Universal Robots URScript: faichun_9jan_1.script

def faichun_9jan_1():
  set_target_payload(1.070000, [0.002000, 0.003000, 0.057000], [0.001723, 0.001723, 0.001723, 0.000000, 0.000000, 0.000000])
  set_tcp(p[0.0,0.0,0.0,0.0,0.0,0.0])
  set_tool_communication(True, 1000000, 2, 1, 1.5, 3.5)
  set_tool_output_mode(0)
  set_tool_digital_output_mode(0, 1)
  set_tool_digital_output_mode(1, 1)
  set_tool_voltage(24)
  step_count_5365f4e1_2aa6_4e7d_952d_8f9d08daece7 = 0.0
  thread Step_Counter_Thread_19057cb8_9120_4cdd_987b_3fe53dc553a4():
    while (True):
      step_count_5365f4e1_2aa6_4e7d_952d_8f9d08daece7 = step_count_5365f4e1_2aa6_4e7d_952d_8f9d08daece7 + 1.0
      sync()
    end
  end
  run Step_Counter_Thread_19057cb8_9120_4cdd_987b_3fe53dc553a4()
  set_safety_mode_transition_hardness(1)
  set_standard_analog_input_domain(0, 1)
  set_standard_analog_input_domain(1, 1)
  set_tool_analog_input_domain(0, 1)
  set_tool_analog_input_domain(1, 1)
  set_analog_outputdomain(0, 0)
  set_analog_outputdomain(1, 0)
  set_input_actions_to_default()
  set_gravity([0.0, 0.0, 9.82])
  global B1empty=False
  global A2Empty=0
  global A1Empty=0
  global B2Empty=False
  global pallet_step=0
  global bright_box=0
  global Pallet_1_cnt=2
  global dark_boxes=0
  global Point_1=p[0.6913645118948067,-0.12399382748223003,0.49223711947071,-1.2983729986843258,1.1259514972191385,-1.2203503861141718]
  # begin: URCap Installation Node
  #   Source: External Control, 1.0.5, FZI Research Center for Information Technology
  #   Type: External Control
  # end: URCap Installation Node
  # begin: URCap Installation Node
  #   Source: OnRobot, 6.2.0, OnRobot A/S
  #   Type: OnRobot Setup
  sleep(1)
  if (False):
  end
  ON_CONN_SHIFT_BOOL = 64
  ON_CONN_SHIFT_INT = 24
  ON_CONN_SHIFT_FLOAT = 24
  ON_CONN_REG_SUM_BOOL = 0
  ON_CONN_REG_SUM_INT = 1
  ON_CONN_REG_SUM_FLOAT = 0
  ON_TOOL_SHIFT_BOOL = 64
  ON_TOOL_SHIFT_INT = 25
  ON_TOOL_SHIFT_FLOAT = 24
  ON_TOOL_SHIFT_BOOL_ARR = [64, 64, 64]
  ON_TOOL_SHIFT_INT_ARR = [25, 25, 25]
  ON_TOOL_SHIFT_FLOAT_ARR = [24, 24, 24]
  ON_TOOL_REG_SUM_BOOL = 0
  ON_TOOL_REG_SUM_INT = 0
  ON_TOOL_REG_SUM_FLOAT = 0
  ON_REGISTERS_SPEEDL_FLOAT = 0
  ON_REG_USE_TOOL = False
  ON_DI_SINGLE = 0
  ON_DI_PRIMARY = 1
  ON_DI_SECONDARY = 2
  ON_DI_DUAL = 3
  on_robot_type = 10
  on_robot_cycle = 2.0
  on_conn_ip = "localhost"
  on_tool_ip = "localhost"
  on_device_socket_port = 51234
  on_conn_xmlrpc = rpc_factory("xmlrpc", "http://localhost:41414")
  on_tool_xmlrpc = rpc_factory("xmlrpc", "http://localhost:41414")
  on_RPC = rpc_factory("xmlrpc", "http://127.0.0.1:31416")
  ON_DEBUG_LOG = False
  on_isMetric = True
  on_toolConnector = True
  on_ioqc = False
  on_dual = False
  on_computebox = False
  on_devices = 0
  on_gripper = [False, False, False]
  on_custom_tcp_id = "none"
  on_custom_tcp_enabled = False
  speedlTime = 0.001
  on_ft = False
  #======    OnRobot Globals    ======#

  ON_MATH_PI=3.141593
  ON_ZEROPOSE=p[0.0,0.0,0.0,0.0,0.0,0.0]
  ON_ZEROFRAME=p[0.0,0.0,0.0,0.0,0.0,0.0]
  ON_ZERO3D=[0.0,0.0,0.0]
  ON_ZERO6D=[0.0,0.0,0.0,0.0,0.0,0.0]
  ON_ZERO8D=[0.0,0.0,0.0,0.0,0.0,0.0,0.0,0.0]
  ON_FALSE3D=[False,False,False]
  ON_FALSE6D=[False,False,False,False,False,False]
  ON_FALSE8D=[False,False,False,False,False,False,False,False]
  global on_return=0
  on_speedL=ON_ZERO6D
  on_speedBase=ON_ZERO6D
  on_speedVect=ON_ZERO6D
  on_speedExtra=ON_ZERO6D
  on_speedCB=ON_ZERO6D
  on_speedGecko=ON_ZERO6D
  on_RTDE_error=0
  on_RTDE_tool_error=0
  on_dataProcess_thrd=0
  ON_DEVICE_ID_MISSING=0
  ON_INIT_WATCHDOG_HZ=5
  ON_INIT_TIMEOUT=2000
  on_robot_TCP_offset=ON_ZEROFRAME
  on_tcp_offset_actual=ON_ZEROFRAME
  on_cog_actual=ON_ZEROFRAME
  on_mass_actual=0.0
  on_robot_mount=[0.0,0.0]

  #======    End of OnRobot Globals    ======#
  #======    OnRobot Interface Messages    ======#

  on_devices_primary_log="OnRobot Devices"
  on_devices_secondary_log="OnRobot Secondary Device"
  on_program_halted="<br>Program halted."
  on_device_error_title="OnRobot - Device error"
  on_install_error="OnRobot Setup is not correct.<br>Check the status in the OnRobot Setup page in the Installation Tab.<br>Program halted."
  on_device_missing="No device connected.<br>Program halted."
  cb_device_missing="No OnRobot Compute Box connected.<br>Program halted."
  ft_device_missing="No OnRobot FT sensor or license detected.<br>Program halted."
  hex_device_missing="No HEX sensor connected.<br>Program halted."
  rg2ft_device_missing="No RG2-FT gripper connected.<br>Program halted."
  rg_device_missing="No RG gripper connected.<br>Program halted."
  vg_device_missing="No VG gripper connected.<br>Program halted."
  gg_device_missing="No Gecko Gripper connected.<br>Program halted."
  sg_device_missing="No Soft Gripper connected.<br>Program halted."
  tfg_device_missing="No 3FG gripper connected.<br>Program halted."
  sdr_device_missing="No OnRobot Sander connected.<br>Program halted."
  twofg_device_missing="No 2FG gripper connected.<br>Program halted."
  vgp_device_missing="No VGP gripper connected.<br>Program halted."
  mg_device_missing="No Magnetic Gripper connected.<br>Program halted."
  fgp_device_missing="No 2FGP20 Gripper connected.<br>Program halted."
  eyes_device_missing="No OnRobot Eyes connected.<br>Program halted."
  on_xmlrpc_start_ip="Connecting to OnRobot XML-RPC Server:"
  on_java_comm_error_textmsg_title="OnRobot - Communication error:"
  on_java_comm_controlsocket_open_error="Socket 'javaSocket' opening was unsuccessful."
  on_java_comm_error_title="OnRobot - Communication error"
  on_java_comm_socket_open_error="Establishing connection with the URCap was timed out.<br>Check the status in the OnRobot Setup page in the Installation Tab.<br>Program halted."
  on_rtde_feed_error_textmsg_title="OnRobot - RTDE error:"
  on_rtde_feed_error="RTDE feed error. OnRobot device count mismatch.<br>Program halted."
  on_rtde_feed_tool_error="Tool RTDE feed error. OnRobot device count mismatch.<br>Program halted."
  on_rtde_feed_open_error_textmsg="Socket 'rtdeFeed' opening was unsuccessful."
  on_rtde_feed_error_title="OnRobot - RTDE error"
  on_rtde_feed_count_error="Invalid RTDE offset setup detected. Please check RTDE Offsets at the OnRobot Setup page in the Installation Tab.<br>Program halted."
  on_rtde_feed_open_error="Establishing connection with the devices was timed out.<br>Ensure that the OnRobot devices are operational, and check the status in the OnRobot Setup page in the Installation Tab."

  #======    End of OnRobot Interface Messages    ======#
  #======    OnRobot Interface    ======#

  on_portopened_javaSocket=False
  on_rtde_feed_opened=False
  on_dataProcess_running=False
  def on_missing():
  popup(on_device_missing,title=on_device_error_title,error=True,blocking=False)
  halt
  end
  def cb_missing():
  popup(cb_device_missing,title=on_device_error_title,error=True,blocking=False)
  halt
  end
  def ft_missing():
  popup(ft_device_missing,title=on_device_error_title,error=True,blocking=False)
  halt
  end
  def hex_missing():
  popup(hex_device_missing,title=on_device_error_title,error=True,blocking=False)
  halt
  end
  def rg2ft_missing():
  popup(rg2ft_device_missing,title=on_device_error_title,error=True,blocking=False)
  halt
  end
  def rg_missing():
  popup(rg_device_missing,title=on_device_error_title,error=True,blocking=False)
  halt
  end
  def vg_missing():
  popup(vg_device_missing,title=on_device_error_title,error=True,blocking=False)
  halt
  end
  def gg_missing():
  popup(gg_device_missing,title=on_device_error_title,error=True,blocking=False)
  halt
  end
  def sg_missing():
  popup(sg_device_missing,title=on_device_error_title,error=True,blocking=False)
  halt
  end
  def tfg_missing():
  popup(tfg_device_missing,title=on_device_error_title,error=True,blocking=False)
  halt
  end
  def sdr_missing():
  popup(sdr_device_missing,title=on_device_error_title,error=True,blocking=False)
  halt
  end
  def twofg_missing():
  popup(twofg_device_missing,title=on_device_error_title,error=True,blocking=False)
  halt
  end
  def vgp_missing():
  popup(vgp_device_missing,title=on_device_error_title,error=True,blocking=False)
  halt
  end
  def mg_missing():
  popup(mg_device_missing,title=on_device_error_title,error=True,blocking=False)
  halt
  end
  def fgp_missing():
  popup(fgp_device_missing,title=on_device_error_title,error=True,blocking=False)
  halt
  end
  def eyes_missing():
  popup(eyes_device_missing,title=on_device_error_title,error=True,blocking=False)
  halt
  end
  def on_portclose_javaSocket():
  socket_close("javaSocket")
  on_portopened_javaSocket=False
  end
  def on_portopen_javaSocket():
  on_portclose_javaSocket()
  on_portopened_javaSocket=socket_open("127.0.0.1",44005,"javaSocket")
  if not on_portopened_javaSocket:
  textmsg(on_java_comm_error_textmsg_title,on_java_comm_controlsocket_open_error)
  popup(on_java_comm_socket_open_error,title=on_java_comm_error_title,error=True,blocking=False)
  halt
  end
  end
  on_conn_rtde_feed_name="rtdeFeedConn"
  on_tool_rtde_feed_name="rtdeFeedTool"
  def on_rtde_feed_close(rtdeFeedName):
  socket_close(rtdeFeedName)
  on_rtde_feed_opened=False
  end
  def on_rtde_feed_open(deviceIP,rtdeFeedName,regStart,regSum,regSpeedl):
  on_rtde_feed_close(rtdeFeedName)
  if((regStart[0]+regSum[0])>128)or((regStart[1]+regSum[1])>48)or((regStart[2]+regSum[2])>48):
  popup(on_rtde_feed_count_error,title=on_rtde_feed_error_title,error=True,blocking=False)
  textmsg(str_cat("RegStart: ",regStart),str_cat("  -  RegSum: ",regSum))
  halt
  end
  on_rtde_feed_opened=socket_open(deviceIP,on_device_socket_port,rtdeFeedName)
  if not on_rtde_feed_opened:
  on_rtde_feed_opened=socket_open(deviceIP,on_device_socket_port,rtdeFeedName)
  end
  if not on_rtde_feed_opened:
  textmsg(on_rtde_feed_error_textmsg_title,on_rtde_feed_open_error_textmsg)
  popup(on_rtde_feed_open_error,title=on_rtde_feed_error_title,error=True,blocking=False)
  halt
  end
  socket_send_int(regStart[0],rtdeFeedName)
  socket_send_int(regSum[0],rtdeFeedName)
  socket_send_int(regStart[1],rtdeFeedName)
  socket_send_int(regSum[1],rtdeFeedName)
  socket_send_int(regStart[2],rtdeFeedName)
  socket_send_int(regSum[2],rtdeFeedName)
  socket_send_int(regSpeedl,rtdeFeedName)
  socket_send_int(on_devices,rtdeFeedName)
  end
  def on_dataRead():
  enter_critical
  on_RTDE_error=read_input_integer_register(ON_CONN_SHIFT_INT)
  if(ON_REG_USE_TOOL):
  on_RTDE_tool_error=read_input_integer_register(ON_TOOL_SHIFT_INT_ARR[0])
  end
  exit_critical
  end
  def on_set_rtde_watchdog(updateHz=ON_INIT_WATCHDOG_HZ):
  local effect="stop"
  if(updateHz<1):
  effect="ignore"
  end
  watchdog_conn_reg_str=str_cat("input_int_register_",ON_CONN_SHIFT_INT)
  rtde_set_watchdog(watchdog_conn_reg_str,updateHz,effect)
  if(ON_REG_USE_TOOL):
  watchdog_tool_reg_str=str_cat("input_int_register_",ON_TOOL_SHIFT_INT_ARR[0])
  rtde_set_watchdog(watchdog_tool_reg_str,updateHz,effect)
  end
  if ON_DEBUG_LOG:
  local update_str=str_cat(" "+effect+" watchdog set to [Hz]: ",updateHz)
  textmsg(watchdog_conn_reg_str,update_str)
  if(ON_REG_USE_TOOL):
  local update_str=str_cat(" "+effect+" watchdog set to [Hz]: ",updateHz)
  textmsg(watchdog_tool_reg_str,update_str)
  end
  end
  end
  def on_speedCB_get():
  return[on_speedCB[0],on_speedCB[1],on_speedCB[2],on_speedCB[3],on_speedCB[4],on_speedCB[5]]
  end
  def on_speedGecko_get():
  local speedExtra=ON_ZERO6D
  if on_speedl_for_gecko:
  speedExtra=[on_speedGecko[0],on_speedGecko[1],on_speedGecko[2],on_speedGecko[3],on_speedGecko[4],on_speedGecko[5]]
  end
  return speedExtra
  end
  def on_speedGecko_set(speedGecko):
  on_speedGecko=[speedGecko[0],speedGecko[1],speedGecko[2],speedGecko[3],speedGecko[4],speedGecko[5]]
  end
  thread on_dataProcess_thread():
  if ON_DEBUG_LOG:
  textmsg("Starting on_dataRead thread")
  end
  local error=False
  on_dataProcess_running=True
  sync()
  while on_dataProcess_running:
  sync()
  on_dataRead()
  error=on_error((on_RTDE_error<0),on_rtde_feed_error,on_rtde_feed_error_title,error)
  error=on_error((ON_REG_USE_TOOL and(on_RTDE_tool_error<0)),on_rtde_feed_tool_error,on_rtde_feed_error_title,error)
  on_dataProcess_running=not error
  end
  if error:
  halt
  end
  if ON_DEBUG_LOG:
  textmsg("Stopping on_dataRead thread")
  end
  end
  thread on_set_watchdog_thread():
  sleep(2)
  on_set_rtde_watchdog(updateHz=ON_INIT_WATCHDOG_HZ)
  sleep(1/ON_INIT_WATCHDOG_HZ)
  on_dataProcess_running=False
  kill on_dataProcess_thrd
  end

  #======    End of OnRobot Interface    ======#
  #======    OnRobot QC Setup Tool Connector    ======#

  def tc_setup_tool():
  if ON_DEBUG_LOG:
  textmsg("QC Setup Tool Connector start...")
  end
  set_tool_voltage(24)

  set_tool_communication(True,1000000,2,1,1.5,3.5)

  if ON_DEBUG_LOG:
  textmsg("QC Setup Tool Connector end.")
  end
  end

  #======    End of OnRobot QC Setup Tool Connector    ======#
  #======    OnRobot TCP Messages    ======#

  on_tcp_log_msg_default="OnRobot: Robot TCP Offset set to:"
  on_tcp_log_msg_primary="OnRobot: Robot TCP Offset set to Primary:"
  on_tcp_log_msg_secondary="OnRobot: Robot TCP Offset set to Secondary:"

  #======    End of OnRobot TCP Messages    ======#
  #======    OnRobot TCP    ======#

  on_tcp_offset_actual=ON_ZEROFRAME
  on_tcp_offset_primary=ON_ZEROFRAME
  on_tcp_static_primary=ON_ZEROFRAME
  on_tcp_dynamic_primary=ON_ZEROFRAME
  on_tcp_adapters=ON_ZEROFRAME
  on_tcp_qc_primary=ON_ZEROFRAME
  on_tcp_base_primary=ON_ZEROFRAME
  on_tcp_gripper_static_primary=ON_ZEROFRAME
  on_tcp_workpiece_primary=ON_ZEROFRAME
  on_tcp_gripper_dynamic_primary=ON_ZEROFRAME
  on_tcp_gripper_primary=ON_ZEROFRAME
  on_tcp_offset_secondary=ON_ZEROFRAME
  on_tcp_static_secondary=ON_ZEROFRAME
  on_tcp_dynamic_secondary=ON_ZEROFRAME
  on_tcp_qc_secondary=ON_ZEROFRAME
  on_tcp_base_secondary=ON_ZEROFRAME
  on_tcp_gripper_static_secondary=ON_ZEROFRAME
  on_tcp_workpiece_secondary=ON_ZEROFRAME
  on_tcp_gripper_dynamic_secondary=ON_ZEROFRAME
  on_tcp_gripper_secondary=ON_ZEROFRAME
  on_tcp_custom_preset_assigned=False
  on_tcp_custom_preset=ON_ZEROFRAME
  def on_tcp_init_adapters():
  if ON_DEBUG_LOG:
  textmsg("TCP Init Adapters start..")
  end
  enter_critical
  on_tcp_adapters=ON_ZEROFRAME
  local adapterCount=length(on_tcp_adapters_array)
  local i=0
  while(i<adapterCount):
  on_tcp_adapters=pose_trans(on_tcp_adapters,on_tcp_adapters_array[i])
  i=i+1
  end
  exit_critical
  if ON_DEBUG_LOG:
  textmsg("TCP Init Adapters end.")
  end
  end
  def on_tcp_update_primary():
  if ON_DEBUG_LOG:
  textmsg("TCP Update Primary start..")
  end
  on_tcp_gripper_dynamic_primary=p[0.0, 0.0, 0.0, 0.0, 0.0, 0.0]
  enter_critical
  on_tcp_dynamic_primary=pose_trans(on_tcp_static_primary,on_tcp_gripper_dynamic_primary)
  on_tcp_offset_primary=pose_trans(on_tcp_dynamic_primary,on_tcp_workpiece_primary)
  exit_critical
  if ON_DEBUG_LOG:
  textmsg("TCP Update Primary end.")
  end
  end
  def on_tcp_init_primary():
  if ON_DEBUG_LOG:
  textmsg("TCP Init Primary start..")
  end
  enter_critical
  on_tcp_base_primary=pose_trans(on_tcp_adapters,on_tcp_qc_primary)
  on_tcp_static_primary=pose_trans(on_tcp_base_primary,on_tcp_gripper_static_primary)
  exit_critical
  on_tcp_update_primary()
  if ON_DEBUG_LOG:
  textmsg("TCP Init Primary end.")
  end
  end
  def on_tcp_offset_set(TCP_offset):
  if ON_DEBUG_LOG:
  textmsg("TCP Offset set started!")
  end
  on_tcp_offset_send(TCP_offset)
  if(on_follow_tcp):
  set_tcp(TCP_offset)
  end
  on_robot_TCP_offset=TCP_offset
  if ON_DEBUG_LOG:
  textmsg("TCP Offset set to: ",on_robot_TCP_offset)
  end
  end
  def on_tcp_offset_forced_set_actual(isPrimary=True):
  if(not on_follow_tcp):

  local tcp_log_msg=on_tcp_log_msg_default

  textmsg(tcp_log_msg,on_tcp_offset_actual)
  set_tcp(on_tcp_offset_actual)
  end
  end
  def on_tcp_update(isPrimary=True):
  on_tcp_update_primary()

  on_tcp_set_actual_to(isPrimary)
  end
  def on_tcp_set_actual_to(isPrimary=True):

  on_tcp_offset_actual=on_tcp_offset_primary
  if(on_follow_tcp):
  textmsg(on_tcp_log_msg_default,on_tcp_offset_actual)
  end

  on_tcp_active_is_primary=isPrimary
  on_tcp_offset_set(on_tcp_offset_actual)
  end
  def on_tcp_update_workpiece_primary(workpiece_offset):
  if ON_DEBUG_LOG:
  textmsg("TCP Update Tool Primary start..")
  end
  on_tcp_workpiece_primary=workpiece_offset
  on_tcp_update_primary()
  if ON_DEBUG_LOG:
  textmsg("TCP Update Tool Primary end.")
  end
  end
  def on_tcp_workpiece_rpy_get(xyz=[0.0,0.0,0.0],rpy=[0.0,0.0,0.0]):
  local rotvec=rpy2rotvec(rpy)
  local workpiece_offset=p[xyz[0],xyz[1],xyz[2],rotvec[0],rotvec[1],rotvec[2]]
  return workpiece_offset
  end

  def on_tcp_update_workpiece(workpiece_offset,tool_index=0):
  if ON_DEBUG_LOG:
  textmsg("TCP Update Tool start..")
  end
  if(tool_index!=ON_DI_SECONDARY):
  on_tcp_update_workpiece_primary(workpiece_offset)
  local isPrimary=True

  end
  on_tcp_set_actual_to(isPrimary)
  if ON_DEBUG_LOG:
  textmsg("TCP Update Tool end.")
  end
  end
  def on_get_tcp_for(tool_index):
  if tool_index==ON_DI_SECONDARY:
  local actual_tcp=on_tcp_static_secondary
  else:
  local actual_tcp=on_tcp_static_primary
  end
  return actual_tcp
  end
  def on_tcp_custom_unused():
  return ON_ZEROFRAME
  end
  def on_tcp_update_custom():
  if ON_DEBUG_LOG:
  textmsg("TCP Update Custom start..")
  end
  if(on_custom_tcp_enabled):
  on_tcp_custom_unused()
  on_tcp_custom_unused()
  on_tcp_custom_unused()
  on_tcp_custom_unused()

  end
  if ON_DEBUG_LOG:
  textmsg("TCP Update Custom end.")
  end
  end

  #======    End of OnRobot TCP    ======#
  #======    OnRobot Payload Messages    ======#

  on_mass_log_msg="OnRobot: Robot Payload Mass set to:"
  on_cog_log_msg="OnRobot: Robot Payload Center of Gravity set to:"

  #======    End of OnRobot Payload Messages    ======#
  #======    OnRobot Payload    ======#

  on_cog_actual=ON_ZEROFRAME
  on_mass_actual=0.0
  on_cog_primary=ON_ZEROFRAME
  on_cog_L1L2_primary=ON_ZEROFRAME
  on_mass_primary=0.0
  on_mass_L1L2_primary=0.0
  on_cog_adapters=ON_ZEROFRAME
  on_cog_qc_primary=ON_ZEROFRAME
  on_cog_base_primary=ON_ZEROFRAME
  on_cog_gripper_primary=ON_ZEROFRAME
  on_cog_workpiece_primary=ON_ZEROFRAME
  on_mass_adapters=0.0
  on_mass_qc_primary=0.0
  on_mass_base_primary=0.0
  on_mass_gripper_primary=0.0
  on_mass_workpiece_primary=0.0
  on_cog_secondary=ON_ZEROFRAME
  on_mass_secondary=0.0
  on_cog_gripper_secondary=ON_ZEROFRAME
  on_mass_gripper_secondary=0.0
  on_cog_workpiece_secondary=ON_ZEROFRAME
  on_mass_workpiece_secondary=0.0
  ON_LB2KG001=0.45359237/100
  def on_payload_init_adapters():
  if ON_DEBUG_LOG:
  textmsg("TCP Init Adapters start..")
  end
  enter_critical
  on_cog_adapters=ON_ZEROFRAME
  on_mass_adapters=0.0
  local massLAL0Ratio=0
  local adapterAbsCOG=ON_ZEROFRAME
  local tcp_adapter_offset=ON_ZEROFRAME
  local adapterCount=length(on_tcp_adapters_array)
  local i=0
  while(i<adapterCount):
  on_mass_adapters=on_mass_adapters+on_mass_adapters_array[i]
  if(on_mass_adapters<=0):
  massLAL0Ratio=0
  else:
  massLAL0Ratio=on_mass_adapters_array[i]/on_mass_adapters
  end
  adapterAbsCOG=pose_trans(tcp_adapter_offset,on_tcp_adapters_array[i])
  adapterAbsCOG=p[adapterAbsCOG[0],adapterAbsCOG[1],adapterAbsCOG[2],0.0,0.0,0.0]
  on_cog_adapters=interpolate_pose(on_cog_adapters,adapterAbsCOG,massLAL0Ratio)
  on_cog_adapters=p[on_cog_adapters[0],on_cog_adapters[1],on_cog_adapters[2],0.0,0.0,0.0]
  tcp_adapter_offset=pose_trans(tcp_adapter_offset,on_tcp_adapters_array[i])
  i=i+1
  sync()
  end
  exit_critical
  if ON_DEBUG_LOG:
  textmsg("TCP Init Adapters end.")
  end
  end
  def on_payload_update_primary():
  if ON_DEBUG_LOG:
  textmsg("Payload Update Primary start..")
  end
  enter_critical
  on_mass_primary=on_mass_L1L2_primary+on_mass_workpiece_primary
  local massL1L2L3Ratio=on_mass_workpiece_primary/on_mass_primary
  local workpieceAbsCOG=pose_trans(on_tcp_dynamic_primary,on_cog_workpiece_primary)
  workpieceAbsCOG=p[workpieceAbsCOG[0],workpieceAbsCOG[1],workpieceAbsCOG[2],0.0,0.0,0.0]
  on_cog_primary=interpolate_pose(on_cog_L1L2_primary,workpieceAbsCOG,massL1L2L3Ratio)
  on_cog_primary=p[on_cog_primary[0],on_cog_primary[1],on_cog_primary[2],0.0,0.0,0.0]
  exit_critical
  if ON_DEBUG_LOG:
  textmsg("Payload Update Primary end.")
  end
  end
  def on_payload_init_primary():
  if ON_DEBUG_LOG:
  textmsg("Payload Init Primary start..")
  end
  enter_critical
  on_mass_base_primary=on_mass_adapters+on_mass_qc_primary
  local massL0L1Ratio=on_mass_qc_primary/on_mass_base_primary
  on_mass_L1L2_primary=on_mass_base_primary+on_mass_gripper_primary
  local massL1L2Ratio=on_mass_gripper_primary/on_mass_L1L2_primary
  local qcAbsCOG=pose_trans(on_tcp_adapters,on_cog_qc_primary)
  qcAbsCOG=p[qcAbsCOG[0],qcAbsCOG[1],qcAbsCOG[2],0.0,0.0,0.0]
  on_cog_base_primary=interpolate_pose(on_cog_adapters,qcAbsCOG,massL0L1Ratio)
  on_cog_base_primary=p[on_cog_base_primary[0],on_cog_base_primary[1],on_cog_base_primary[2],0.0,0.0,0.0]
  local gripperAbsCOG=pose_trans(on_tcp_base_primary,on_cog_gripper_primary)
  gripperAbsCOG=p[gripperAbsCOG[0],gripperAbsCOG[1],gripperAbsCOG[2],0.0,0.0,0.0]
  on_cog_L1L2_primary=interpolate_pose(on_cog_base_primary,gripperAbsCOG,massL1L2Ratio)
  on_cog_L1L2_primary=p[on_cog_L1L2_primary[0],on_cog_L1L2_primary[1],on_cog_L1L2_primary[2],0.0,0.0,0.0]
  exit_critical
  on_payload_update_primary()
  if ON_DEBUG_LOG:
  textmsg("Payload Init Primary end.")
  end
  end
  def on_payload_update():
  on_payload_update_primary()

  on_mass_actual =on_mass_primary
  on_cog_actual=on_cog_primary

  on_payload_set_actual()
  end
  def on_payload_set_actual():

  on_mass_actual =on_mass_primary
  on_cog_actual=on_cog_primary

  local CoG=[on_cog_actual[0],on_cog_actual[1],on_cog_actual[2]]
  on_payload_set(on_mass_actual,CoG)
  end
  def on_payload_update_workpiece_primary(workpiece_mass=0,workpiece_cog=[0.0,0.0,0.0]):
  if ON_DEBUG_LOG:
  textmsg("Payload Update Workpiece Primary start..")
  end
  on_cog_workpiece_primary=p[workpiece_cog[0],workpiece_cog[1],workpiece_cog[2],0.0,0.0,0.0]
  on_mass_workpiece_primary=workpiece_mass
  on_payload_update_primary()
  if ON_DEBUG_LOG:
  textmsg("Payload Update Workpiece Primary end.")
  end
  end
  def on_payload_set(mass,CoG):
  if ON_DEBUG_LOG:
  textmsg("Payload set started!")
  end
  local center_of_gravity=[CoG[0],CoG[1],CoG[2]]
  on_payload_send(center_of_gravity,mass)
  if(on_isMetric):
  local roundedMass=floor(mass*100+0.5)/100
  else:
  local roundedMass=floor(mass/ON_LB2KG001+0.5)*ON_LB2KG001
  end
  set_payload(roundedMass,center_of_gravity)
  on_mass_actual=roundedMass
  on_cog_actual=p[CoG[0],CoG[1],CoG[2],0.0,0.0,0.0]
  if ON_DEBUG_LOG:
  textmsg("Payload mass, CoG set to: ",str_cat(str_cat(mass,", "),CoG))
  end
  end

  def on_payload_update_secondary():
  end
  def on_payload_init_secondary():
  end

  def on_payload_update_workpiece(workpiece_mass,workpiece_cog=[0.0,0.0,0.0],tool_index=0):
  if ON_DEBUG_LOG:
  textmsg("Payload Update Workpiece start..")
  end
  if(tool_index!=ON_DI_SECONDARY):
  on_cog_workpiece_primary=p[workpiece_cog[0],workpiece_cog[1],workpiece_cog[2],0.0,0.0,0.0]
  on_mass_workpiece_primary=workpiece_mass
  else:
  on_cog_workpiece_secondary=p[workpiece_cog[0],workpiece_cog[1],workpiece_cog[2],0.0,0.0,0.0]
  on_mass_workpiece_secondary=workpiece_mass
  end
  on_payload_update()
  if ON_DEBUG_LOG:
  textmsg("Payload Update Workpiece end.")
  end
  end
  def on_payload_get_cog2tcp_workpiece(tool_index=0):
  if(tool_index!=ON_DI_SECONDARY):
  local cog_tool=[on_tcp_workpiece_primary[0],on_tcp_workpiece_primary[1],on_tcp_workpiece_primary[2]]
  else:
  local cog_tool=[on_tcp_workpiece_secondary[0],on_tcp_workpiece_secondary[1],on_tcp_workpiece_secondary[2]]
  end
  return cog_tool
  end

  #======    End of OnRobot Payload    ======#
  #======    OnRobot QC TCP    ======#

  onrobotmini=0

  def on_tcp_offset_send(TCP_offset):
  on_robot_TCP_offset=TCP_offset
  end
  def on_payload_send(CoG,mass):
  on_robot_payload_cog=CoG
  on_robot_payload_mass=mass
  end


  #======    End of OnRobot QC TCP    ======#
  #======    OnRobot  Speedl    ======#

  on_speedl_thread_handler=0
  on_speedl_is_enabled=False
  on_speedl_is_running=False
  on_speedl_acc=0.0
  ft_speedl_hg_caranteen_reached=False
  ft_speedl_hg_caranteen_safemode=False
  on_speedl_for_ftcontrol=False
  on_speedl_for_move=False
  on_speedl_for_handguide=False
  on_speedl_for_insertpart=False
  on_speedl_for_depthcompensation=False
  on_speedl_for_center=False
  on_speedl_for_gecko=False
  on_speedl_acc=10000.0
  on_speedl_acc_to_zero=3.0
  ON_SPEEDL_FTCONTROL=1
  ON_SPEEDL_HANDGUIDE=2
  ON_SPEEDL_TRAJECTORY=3
  ON_SPEEDL_MOVE=ON_SPEEDL_TRAJECTORY
  ON_SPEEDL_INSERTPART=4
  ON_SPEEDL_DEPTHCOMP=5
  ON_SPEEDL_CENTER=6
  ON_SPEEDL_GECKO=7
  def on_wait_ms(time_ms):
  local sync_time=ceil(norm(time_ms/2.0))
  while(sync_time>0):
  sync_time=sync_time-1
  sync()
  end
  end
  def on_error(status_flag,message,title,stop_var=False):
  if(status_flag):
  popup(message,title=title,error=True,blocking=False)
  stop_var=True
  end
  return stop_var
  end
  def on_warning(status_flag,message,title,isPopupNeeded=False,is_shown=False):
  if(status_flag):
  if(not is_shown):
  if(isPopupNeeded):
  popup(message,title=title,warning=True,blocking=False)
  else:
  textmsg(title+": ",message)
  end
  is_shown=True
  end
  else:
  is_shown=False
  end
  return is_shown
  end
  def on_speedl_add_extra(speedBase,speedExtra):
  speedSum=ON_ZERO6D
  speedBaseP=p[speedBase[0],speedBase[1],speedBase[2],speedBase[3],speedBase[4],speedBase[5]]
  speedExtraP=p[speedExtra[0],speedExtra[1],speedExtra[2],speedExtra[3],speedExtra[4],speedExtra[5]]
  speedSumP=pose_add(speedExtraP,speedBaseP)
  speedSum=[speedSumP[0],speedSumP[1],speedSumP[2],speedSumP[3],speedSumP[4],speedSumP[5]]
  return speedSum
  end

  thread on_speedl_thread():
  if ON_DEBUG_LOG:
  textmsg("Speedl thread started..")
  end
  enter_critical
  on_speedl_is_running=True
  on_speedl_is_enabled=True
  exit_critical
  on_speedL=ON_ZERO6D
  on_speedL_last=ON_ZERO6D

  while on_speedl_is_running:
  on_speedBase=on_speedCB_get()
  on_speedL=on_speedBase


  if on_speedl_is_enabled:
  if(on_speedL==ON_ZERO6D):
  on_speedL=[on_speedL_last[0]/100,on_speedL_last[1]/100,on_speedL_last[2]/100,on_speedL_last[3]/100,on_speedL_last[4]/100,on_speedL_last[5]/100]
  end
  speedl(on_speedL,a=on_speedl_acc,t=speedlTime)
  else:
  speedl(ON_ZERO6D,a=on_speedl_acc_to_zero,t=speedlTime)
  end
  on_speedL_last=on_speedL
  end

  on_speedL=ON_ZERO6D
  if ON_DEBUG_LOG:
  textmsg("Speedl thread ended.")
  end
  end
  def on_speedl_integer_get():
  local speedl_integer=binary_list_to_integer([on_speedl_for_ftcontrol,on_speedl_for_handguide,on_speedl_for_move,on_speedl_for_insertpart,on_speedl_for_depthcompensation,on_speedl_for_center,on_speedl_for_gecko])
  return speedl_integer
  end
  def on_speedl_start_for(speedl_id):
  if(speedl_id==ON_SPEEDL_FTCONTROL):
  on_speedl_for_ftcontrol=True
  elif(speedl_id==ON_SPEEDL_HANDGUIDE):
  on_speedl_for_handguide=True
  elif(speedl_id==ON_SPEEDL_TRAJECTORY):
  on_speedl_for_move=True
  elif(speedl_id==ON_SPEEDL_INSERTPART):
  on_speedl_for_insertpart=True
  elif(speedl_id==ON_SPEEDL_DEPTHCOMP):
  on_speedl_for_depthcompensation=True
  elif(speedl_id==ON_SPEEDL_CENTER):
  on_speedl_for_center=True
  elif(speedl_id==ON_SPEEDL_GECKO):
  on_speedl_for_gecko=True
  else:
  textmsg("Unknown Start speedl ID received: ",speedl_id)
  end
  local speedl_integer=on_speedl_integer_get()
  if not(speedl_integer==0):
  if not on_speedl_is_running:
  on_speedl_thread_handler=run on_speedl_thread()
  end
  end
  return on_speedl_is_running
  end
  def on_speedl_stop_for(speedl_id,brake=10,brakeRot=10):
  if(speedl_id==ON_SPEEDL_FTCONTROL):
  on_speedl_for_ftcontrol=False
  elif(speedl_id==ON_SPEEDL_HANDGUIDE):
  on_speedl_for_handguide=False
  elif(speedl_id==ON_SPEEDL_TRAJECTORY):
  on_speedl_for_move=False
  elif(speedl_id==ON_SPEEDL_INSERTPART):
  on_speedl_for_insertpart=False
  elif(speedl_id==ON_SPEEDL_DEPTHCOMP):
  on_speedl_for_depthcompensation=False
  elif(speedl_id==ON_SPEEDL_CENTER):
  on_speedl_for_center=False
  elif(speedl_id==ON_SPEEDL_GECKO):
  on_speedl_for_gecko=False
  on_speedGecko_set(ON_ZERO6D)
  else:
  textmsg("Unknown Stop speedl ID received: ",speedl_id)
  end
  local speedl_integer=on_speedl_integer_get()
  if(speedl_integer==0):
  if(on_speedl_is_running):
  kill on_speedl_thread_handler
  enter_critical
  on_speedl_is_running=False
  exit_critical

  end
  if ON_DEBUG_LOG:
  textmsg("Speedl thread stopped")
  end
  stopl(brake,brakeRot)
  end
  return on_speedl_is_running
  end
  def on_speedl_pause():
  on_speedl_is_enabled=False
  return on_speedl_integer_get()
  end
  def on_speedl_resume():
  on_speedl_is_enabled=True
  return on_speedl_integer_get()
  end

  #======    End of OnRobot  Speedl    ======#
  textmsg(on_devices_primary_log, ": Quick Changer + QC Tool Side + [0.0, 0.0, 0.0, 0.0, 0.0, 0.0]")
  on_follow_tcp = False
  on_tcp_active_is_primary = True
  on_tcp_adapters_array = []
  on_cog_adapters_array = []
  on_mass_adapters_array = []
  on_tcp_qc_primary = p[0.0, 0.0, 0.0136, 0.0, 0.0, 0.0]
  on_cog_qc_primary = p[0.0, 0.0, 0.004, 0.0, 0.0, 0.0]
  on_mass_qc_primary = 0.06
  on_tcp_gripper_static_primary = p[0.0, 0.0, 0.017, 0.0, 0.0, 0.0]
  on_cog_gripper_primary = p[0.0, 0.0, 0.002, 0.0, 0.0, 0.0]
  on_mass_gripper_primary = 0.14
  on_tcp_workpiece_primary = p[0.0, 0.0, 0.0, 0.0, 0.0, 0.0]
  on_cog_workpiece_primary = p[0.0, 0.0, 0.0, 0.0, 0.0, 0.0]
  on_mass_workpiece_primary = 0.0
  #======    OnRobot Run    ======#

  on_portopen_javaSocket()
  sync()
  textmsg(on_xmlrpc_start_ip,on_conn_ip)
  if(ON_REG_USE_TOOL):
  on_regStart_conn=[ON_CONN_SHIFT_BOOL,ON_CONN_SHIFT_INT,ON_CONN_SHIFT_FLOAT]
  on_regSum_conn=[ON_CONN_REG_SUM_BOOL,ON_CONN_REG_SUM_INT,ON_CONN_REG_SUM_FLOAT]
  on_rtde_feed_open(on_conn_ip,on_conn_rtde_feed_name,on_regStart_conn,on_regSum_conn,ON_REGISTERS_SPEEDL_FLOAT)
  sync()
  textmsg(on_xmlrpc_start_ip,on_tool_ip)
  on_regStart_tool=[ON_TOOL_SHIFT_BOOL,ON_TOOL_SHIFT_INT,ON_TOOL_SHIFT_FLOAT]
  on_regSum_tool=[ON_TOOL_REG_SUM_BOOL,ON_TOOL_REG_SUM_INT,ON_TOOL_REG_SUM_FLOAT]
  on_rtde_feed_open(on_tool_ip,on_tool_rtde_feed_name,on_regStart_tool,on_regSum_tool,0)
  sync()
  else:
  on_regStart_conn=[ON_CONN_SHIFT_BOOL,ON_CONN_SHIFT_INT,ON_CONN_SHIFT_FLOAT]
  on_regSum_conn=[ON_CONN_REG_SUM_BOOL,ON_CONN_REG_SUM_INT,ON_CONN_REG_SUM_FLOAT]
  on_rtde_feed_open(on_conn_ip,on_conn_rtde_feed_name,on_regStart_conn,on_regSum_conn,ON_REGISTERS_SPEEDL_FLOAT)
  sync()
  end
  on_set_rtde_watchdog(updateHz=0.2)
  sync()
  on_dataProcess_thrd=run on_dataProcess_thread()
  sync()
  on_tcp_init_adapters()
  on_payload_init_adapters()
  on_tcp_init_primary()
  on_payload_init_primary()

  on_tcp_update_custom()
  on_tcp_set_actual_to(on_tcp_active_is_primary)
  if(on_follow_tcp):
  on_payload_set_actual()
  end
  on_watchdog_thrd=run on_set_watchdog_thread()
  sync()
  def done_waiting_for_init(device_name,product_code,tool_index=0):
  textmsg(str_cat(device_name,str_cat(str_cat("[",tool_index),"]: ")),product_code)
  end

  #======    End of OnRobot Run    ======#
  #======    OnRobot QC Start    ======#

  if(on_toolConnector):
  tc_setup_tool()
  end
  sync()

  #======    End of OnRobot QC Start    ======#
  # end: URCap Installation Node
  $ 1 "Robot Program"
  $ 2 "Script: FaiChun_9 Jan_11_2.script"
  def Machining1():
    # Default parameters:
    global speed_ms = 0.05
    global speed_rads = 0.75
    global accel_mss = 3
    global accel_radss = 1.2
    global blend_radius_m = 0.0003

    # Add subprograms here
    # Start of main program
    # Program generated by RoboDK v5.6.8 for UR10e on 14/01/2025 11:38:46
    # Using nominal kinematics.
    blend_radius_m = 0.0003
    speed_ms = 0.05
    # set_reference(p[0.340000, -0.055000, 0.001500, 0.000000, 0.000000, 0.000000])
    set_tcp(p[0.000000, 0.000000, 0.252000, 0.000000, 0.000000, 0.000000])
    # Show Tool
    movej([0.533483, -1.384929, -2.455828, -0.871632, 1.570796, 2.104279],accel_radss,speed_rads,0,blend_radius_m)
    movel([0.533483, -1.438119, -2.486082, -0.788188, 1.570796, 2.104279],accel_mss,speed_ms,0,blend_radius_m)
    #SetTool1
    #M_RunCode6
    #SetRPM60000
    speed_ms = 0.05
    #M_RunCode3
    movel([0.533483, -1.461338, -2.497320, -0.753730, 1.570796, 2.104279],accel_mss,speed_ms,0,blend_radius_m)
    speed_ms = 0.003
    movel([0.533483, -1.467339, -2.500058, -0.744992, 1.570796, 2.104279],accel_mss,speed_ms,0,blend_radius_m)
    speed_ms = 0.02
    movel([0.259918, -1.461630, -2.504809, -0.745950, 1.570796, 1.830715],accel_mss,speed_ms,0,blend_radius_m)
    movel([0.369740, -1.126670, -2.705271, -0.880448, 1.570796, 1.940536],accel_mss,speed_ms,0,blend_radius_m)
    movel([0.742885, -1.140080, -2.699787, -0.872522, 1.570796, 2.313681],accel_mss,speed_ms,0,blend_radius_m)
    movel([0.533483, -1.467339, -2.500058, -0.744992, 1.570796, 2.104279],accel_mss,speed_ms,0,blend_radius_m)
    speed_ms = 0.003
    movel([0.533483, -1.461338, -2.497320, -0.753730, 1.570796, 2.104279],accel_mss,speed_ms,0,blend_radius_m)
    speed_ms = 0.05
    movel([0.533483, -1.438119, -2.486082, -0.788188, 1.570796, 2.104279],accel_mss,speed_ms,0,blend_radius_m)
    #M_RunCode9
    movel([0.533312, -1.429268, -2.493105, -0.790016, 1.570796, 2.104108],accel_mss,speed_ms,0,blend_radius_m)
    #M_RunCode3
    movel([0.533312, -1.452668, -2.504450, -0.755271, 1.570796, 2.104108],accel_mss,speed_ms,0,blend_radius_m)
    speed_ms = 0.003
    movel([0.533312, -1.458718, -2.507214, -0.746458, 1.570796, 2.104108],accel_mss,speed_ms,0,blend_radius_m)
    speed_ms = 0.012
    movel([0.529447, -1.458110, -2.507714, -0.746565, 1.570796, 2.100243],accel_mss,speed_ms,0,blend_radius_m)
    movel([0.527191, -1.462019, -2.504487, -0.745883, 1.570796, 2.097987],accel_mss,speed_ms,0,blend_radius_m)
    movel([0.521465, -1.461157, -2.505201, -0.746031, 1.570796, 2.092261],accel_mss,speed_ms,0,blend_radius_m)
    movel([0.523700, -1.457237, -2.508431, -0.746721, 1.570796, 2.094496],accel_mss,speed_ms,0,blend_radius_m)
    movel([0.521680, -1.456940, -2.508675, -0.746774, 1.570796, 2.092476],accel_mss,speed_ms,0,blend_radius_m)
    movel([0.519450, -1.460862, -2.505444, -0.746082, 1.570796, 2.090246],accel_mss,speed_ms,0,blend_radius_m)
    movel([0.514625, -1.460178, -2.506009, -0.746201, 1.570796, 2.085422],accel_mss,speed_ms,0,blend_radius_m)
    movel([0.513688, -1.460046, -2.506118, -0.746224, 1.570796, 2.084485],accel_mss,speed_ms,0,blend_radius_m)
    movel([0.516966, -1.454221, -2.510901, -0.747267, 1.570796, 2.087762],accel_mss,speed_ms,0,blend_radius_m)
    movel([0.520880, -1.454777, -2.510447, -0.747166, 1.570796, 2.091676],accel_mss,speed_ms,0,blend_radius_m)
    movel([0.522047, -1.452724, -2.512121, -0.747544, 1.570796, 2.092844],accel_mss,speed_ms,0,blend_radius_m)
    movel([0.516087, -1.451882, -2.512806, -0.747701, 1.570796, 2.086883],accel_mss,speed_ms,0,blend_radius_m)
    movel([0.511663, -1.459770, -2.506346, -0.746273, 1.570796, 2.082459],accel_mss,speed_ms,0,blend_radius_m)
    movel([0.510722, -1.459645, -2.506450, -0.746294, 1.570796, 2.081518],accel_mss,speed_ms,0,blend_radius_m)
    speed_ms = 0.02
    movel([0.402251, -1.451333, -2.513252, -0.747803, 1.570796, 1.973047],accel_mss,speed_ms,0,blend_radius_m)
    movel([0.287164, -1.455120, -2.510166, -0.747103, 1.570796, 1.857961],accel_mss,speed_ms,0,blend_radius_m)
    speed_ms = 0.012
    movel([0.289732, -1.447134, -2.516649, -0.748606, 1.570796, 1.860528],accel_mss,speed_ms,0,blend_radius_m)
    movel([0.283110, -1.447719, -2.516177, -0.748493, 1.570796, 1.853907],accel_mss,speed_ms,0,blend_radius_m)
    movel([0.282451, -1.449796, -2.514499, -0.748094, 1.570796, 1.853247],accel_mss,speed_ms,0,blend_radius_m)
    movel([0.286803, -1.449409, -2.514812, -0.748168, 1.570796, 1.857599],accel_mss,speed_ms,0,blend_radius_m)
    movel([0.284916, -1.455306, -2.510014, -0.747069, 1.570796, 1.855712],accel_mss,speed_ms,0,blend_radius_m)
    movel([0.283876, -1.455397, -2.509940, -0.747053, 1.570796, 1.854673],accel_mss,speed_ms,0,blend_radius_m)
    movel([0.278513, -1.455877, -2.509546, -0.746965, 1.570796, 1.849310],accel_mss,speed_ms,0,blend_radius_m)
    movel([0.279756, -1.451908, -2.512785, -0.747696, 1.570796, 1.850552],accel_mss,speed_ms,0,blend_radius_m)
    movel([0.277501, -1.452116, -2.512616, -0.747657, 1.570796, 1.848297],accel_mss,speed_ms,0,blend_radius_m)
    movel([0.276268, -1.456086, -2.509375, -0.746928, 1.570796, 1.847065],accel_mss,speed_ms,0,blend_radius_m)
    movel([0.269859, -1.456703, -2.508870, -0.746817, 1.570796, 1.840655],accel_mss,speed_ms,0,blend_radius_m)
    movel([0.271062, -1.452742, -2.512107, -0.747540, 1.570796, 1.841859],accel_mss,speed_ms,0,blend_radius_m)
    movel([0.266709, -1.453184, -2.511747, -0.747458, 1.570796, 1.837505],accel_mss,speed_ms,0,blend_radius_m)
    movel([0.268482, -1.447281, -2.516530, -0.748577, 1.570796, 1.839278],accel_mss,speed_ms,0,blend_radius_m)
    movel([0.272863, -1.446832, -2.516892, -0.748665, 1.570796, 1.843659],accel_mss,speed_ms,0,blend_radius_m)
    movel([0.273500, -1.444749, -2.518566, -0.749074, 1.570796, 1.844297],accel_mss,speed_ms,0,blend_radius_m)
    movel([0.269110, -1.445198, -2.518206, -0.748985, 1.570796, 1.839906],accel_mss,speed_ms,0,blend_radius_m)
    movel([0.270618, -1.440202, -2.522197, -0.749990, 1.570796, 1.841414],accel_mss,speed_ms,0,blend_radius_m)
    movel([0.270916, -1.439225, -2.522974, -0.750190, 1.570796, 1.841713],accel_mss,speed_ms,0,blend_radius_m)
    movel([0.277462, -1.438552, -2.523507, -0.750330, 1.570796, 1.848259],accel_mss,speed_ms,0,blend_radius_m)
    movel([0.276210, -1.442598, -2.520288, -0.749503, 1.570796, 1.847006],accel_mss,speed_ms,0,blend_radius_m)
    movel([0.278494, -1.442373, -2.520467, -0.749548, 1.570796, 1.849291],accel_mss,speed_ms,0,blend_radius_m)
    movel([0.280415, -1.436214, -2.525356, -0.750819, 1.570796, 1.851211],accel_mss,speed_ms,0,blend_radius_m)
    movel([0.271556, -1.437117, -2.524643, -0.750629, 1.570796, 1.842352],accel_mss,speed_ms,0,blend_radius_m)
    movel([0.309866, -1.316419, -2.609463, -0.786507, 1.570796, 1.880662],accel_mss,speed_ms,0,blend_radius_m)
    speed_ms = 0.02
    movel([0.360938, -1.167682, -2.687935, -0.856771, 1.570796, 1.931735],accel_mss,speed_ms,0,blend_radius_m)
    movel([0.361480, -1.166168, -2.688606, -0.857615, 1.570796, 1.932276],accel_mss,speed_ms,0,blend_radius_m)
    speed_ms = 0.012
    movel([0.373333, -1.164332, -2.689415, -0.858642, 1.570796, 1.944129],accel_mss,speed_ms,0,blend_radius_m)
    movel([0.376888, -1.154641, -2.693631, -0.864117, 1.570796, 1.947684],accel_mss,speed_ms,0,blend_radius_m)
    movel([0.373789, -1.155114, -2.693427, -0.863848, 1.570796, 1.944585],accel_mss,speed_ms,0,blend_radius_m)
    movel([0.371457, -1.161503, -2.690656, -0.860230, 1.570796, 1.942254],accel_mss,speed_ms,0,blend_radius_m)
    movel([0.362659, -1.162880, -2.690053, -0.859456, 1.570796, 1.933456],accel_mss,speed_ms,0,blend_radius_m)
    movel([0.363202, -1.161358, -2.690719, -0.860312, 1.570796, 1.933999],accel_mss,speed_ms,0,blend_radius_m)
    movel([0.366035, -1.153430, -2.694151, -0.864808, 1.570796, 1.936831],accel_mss,speed_ms,0,blend_radius_m)
    movel([0.372034, -1.152469, -2.694563, -0.865358, 1.570796, 1.942830],accel_mss,speed_ms,0,blend_radius_m)
    movel([0.373252, -1.149115, -2.695992, -0.867282, 1.570796, 1.944048],accel_mss,speed_ms,0,blend_radius_m)
    movel([0.367233, -1.150084, -2.695580, -0.866725, 1.570796, 1.938029],accel_mss,speed_ms,0,blend_radius_m)
    movel([0.370700, -1.140431, -2.699641, -0.872317, 1.570796, 1.941496],accel_mss,speed_ms,0,blend_radius_m)
    movel([0.376777, -1.139438, -2.700053, -0.872898, 1.570796, 1.947573],accel_mss,speed_ms,0,blend_radius_m)
    movel([0.379196, -1.132819, -2.702778, -0.876792, 1.570796, 1.949992],accel_mss,speed_ms,0,blend_radius_m)
    movel([0.388243, -1.131390, -2.703361, -0.877639, 1.570796, 1.959039],accel_mss,speed_ms,0,blend_radius_m)
    movel([0.385765, -1.138032, -2.700635, -0.873721, 1.570796, 1.956561],accel_mss,speed_ms,0,blend_radius_m)
    movel([0.388910, -1.137558, -2.700831, -0.873999, 1.570796, 1.959706],accel_mss,speed_ms,0,blend_radius_m)
    movel([0.391408, -1.130908, -2.703557, -0.877924, 1.570796, 1.962205],accel_mss,speed_ms,0,blend_radius_m)
    movel([0.400429, -1.129586, -2.704093, -0.878710, 1.570796, 1.971225],accel_mss,speed_ms,0,blend_radius_m)
    movel([0.396655, -1.139442, -2.700052, -0.872896, 1.570796, 1.967451],accel_mss,speed_ms,0,blend_radius_m)
    movel([0.390623, -1.140304, -2.699694, -0.872391, 1.570796, 1.961419],accel_mss,speed_ms,0,blend_radius_m)
    movel([0.389336, -1.143717, -2.698269, -0.870403, 1.570796, 1.960133],accel_mss,speed_ms,0,blend_radius_m)
    movel([0.398466, -1.142432, -2.698807, -0.871151, 1.570796, 1.969263],accel_mss,speed_ms,0,blend_radius_m)
    movel([0.403585, -1.129142, -2.704273, -0.878974, 1.570796, 1.974381],accel_mss,speed_ms,0,blend_radius_m)
    movel([0.563013, -1.120295, -2.707818, -0.884277, 1.570796, 2.133810],accel_mss,speed_ms,0,blend_radius_m)
    speed_ms = 0.02
    movel([0.707055, -1.139837, -2.699888, -0.872664, 1.570796, 2.277852],accel_mss,speed_ms,0,blend_radius_m)
    movel([0.698676, -1.152794, -2.694424, -0.865172, 1.570796, 2.269473],accel_mss,speed_ms,0,blend_radius_m)
    speed_ms = 0.012
    movel([0.706130, -1.154616, -2.693642, -0.864132, 1.570796, 2.276927],accel_mss,speed_ms,0,blend_radius_m)
    movel([0.708299, -1.151299, -2.695063, -0.866028, 1.570796, 2.279096],accel_mss,speed_ms,0,blend_radius_m)
    movel([0.703392, -1.150081, -2.695581, -0.866727, 1.570796, 2.274188],accel_mss,speed_ms,0,blend_radius_m)
    movel([0.709631, -1.140484, -2.699619, -0.872286, 1.570796, 2.280428],accel_mss,speed_ms,0,blend_radius_m)
    movel([0.710822, -1.140781, -2.699495, -0.872113, 1.570796, 2.281618],accel_mss,speed_ms,0,blend_radius_m)
    movel([0.716930, -1.142343, -2.698844, -0.871202, 1.570796, 2.287726],accel_mss,speed_ms,0,blend_radius_m)
    movel([0.712681, -1.148808, -2.696122, -0.867459, 1.570796, 2.283477],accel_mss,speed_ms,0,blend_radius_m)
    movel([0.715213, -1.149470, -2.695841, -0.867078, 1.570796, 2.286009],accel_mss,speed_ms,0,blend_radius_m)
    movel([0.719478, -1.143013, -2.698564, -0.870812, 1.570796, 2.290274],accel_mss,speed_ms,0,blend_radius_m)
    movel([0.726693, -1.144971, -2.697742, -0.869675, 1.570796, 2.297489],accel_mss,speed_ms,0,blend_radius_m)
    movel([0.722404, -1.151397, -2.695021, -0.865972, 1.570796, 2.293201],accel_mss,speed_ms,0,blend_radius_m)
    movel([0.727224, -1.152737, -2.694448, -0.865204, 1.570796, 2.298021],accel_mss,speed_ms,0,blend_radius_m)
    movel([0.720946, -1.162096, -2.690396, -0.859897, 1.570796, 2.291743],accel_mss,speed_ms,0,blend_radius_m)
    movel([0.716151, -1.160787, -2.690968, -0.860634, 1.570796, 2.286947],accel_mss,speed_ms,0,blend_radius_m)
    movel([0.713986, -1.164044, -2.689542, -0.858803, 1.570796, 2.284782],accel_mss,speed_ms,0,blend_radius_m)
    movel([0.718770, -1.165346, -2.688968, -0.858075, 1.570796, 2.289566],accel_mss,speed_ms,0,blend_radius_m)
    movel([0.713629, -1.173035, -2.685547, -0.853807, 1.570796, 2.284425],accel_mss,speed_ms,0,blend_radius_m)
    movel([0.712640, -1.174516, -2.684881, -0.852992, 1.570796, 2.283436],accel_mss,speed_ms,0,blend_radius_m)
    movel([0.705579, -1.172648, -2.685720, -0.854020, 1.570796, 2.276375],accel_mss,speed_ms,0,blend_radius_m)
    movel([0.709681, -1.166442, -2.688485, -0.857463, 1.570796, 2.280478],accel_mss,speed_ms,0,blend_radius_m)
    movel([0.707181, -1.165792, -2.688772, -0.857825, 1.570796, 2.277978],accel_mss,speed_ms,0,blend_radius_m)
    movel([0.700980, -1.175214, -2.684566, -0.852609, 1.570796, 2.271776],accel_mss,speed_ms,0,blend_radius_m)
    movel([0.710514, -1.177702, -2.683440, -0.851247, 1.570796, 2.281311],accel_mss,speed_ms,0,blend_radius_m)
    speed_ms = 0.02
    movel([0.615153, -1.324265, -2.604567, -0.783557, 1.570796, 2.185950],accel_mss,speed_ms,0,blend_radius_m)
    movel([0.542601, -1.442874, -2.520067, -0.749448, 1.570796, 2.113397],accel_mss,speed_ms,0,blend_radius_m)
    speed_ms = 0.012
    movel([0.534737, -1.441630, -2.521060, -0.749699, 1.570796, 2.105533],accel_mss,speed_ms,0,blend_radius_m)
    movel([0.531216, -1.447708, -2.516186, -0.748495, 1.570796, 2.102013],accel_mss,speed_ms,0,blend_radius_m)
    movel([0.533250, -1.448021, -2.515933, -0.748434, 1.570796, 2.104046],accel_mss,speed_ms,0,blend_radius_m)
    movel([0.535568, -1.444031, -2.519142, -0.749216, 1.570796, 2.106364],accel_mss,speed_ms,0,blend_radius_m)
    movel([0.541367, -1.444954, -2.518401, -0.749033, 1.570796, 2.112164],accel_mss,speed_ms,0,blend_radius_m)
    movel([0.540803, -1.445915, -2.517630, -0.748844, 1.570796, 2.111599],accel_mss,speed_ms,0,blend_radius_m)
    movel([0.537910, -1.450844, -2.513649, -0.747896, 1.570796, 2.108707],accel_mss,speed_ms,0,blend_radius_m)
    movel([0.534018, -1.450225, -2.514152, -0.748013, 1.570796, 2.104814],accel_mss,speed_ms,0,blend_radius_m)
    movel([0.532824, -1.452279, -2.512483, -0.747626, 1.570796, 2.103621],accel_mss,speed_ms,0,blend_radius_m)
    movel([0.536712, -1.452896, -2.511981, -0.747512, 1.570796, 2.107508],accel_mss,speed_ms,0,blend_radius_m)
    movel([0.533312, -1.458718, -2.507214, -0.746458, 1.570796, 2.104108],accel_mss,speed_ms,0,blend_radius_m)
    speed_ms = 0.003
    movel([0.533312, -1.452668, -2.504450, -0.755271, 1.570796, 2.104108],accel_mss,speed_ms,0,blend_radius_m)
    speed_ms = 0.05
    movel([0.533312, -1.429268, -2.493105, -0.790016, 1.570796, 2.104108],accel_mss,speed_ms,0,blend_radius_m)
    #M_RunCode9
    movel([0.417526, -1.170993, -2.652148, -0.889248, 1.570796, 1.988323],accel_mss,speed_ms,0,blend_radius_m)
    #M_RunCode3
    # num 0 inside
    movel([0.417526, -1.198293, -2.666816, -0.847281, 1.570796, 1.988323],accel_mss,speed_ms,0,blend_radius_m)
    speed_ms = 0.003
    movel([0.417526, -1.205477, -2.670419, -0.836494, 1.570796, 1.988323],accel_mss,speed_ms,0,blend_radius_m)
    speed_ms = 0.015
    movel([0.408855, -1.212168, -2.667155, -0.833065, 1.570796, 1.979651],accel_mss,speed_ms,0,blend_radius_m)
    movel([0.402561, -1.216461, -2.665035, -0.830893, 1.570796, 1.973358],accel_mss,speed_ms,0,blend_radius_m)
    movel([0.400243, -1.217697, -2.664421, -0.830271, 1.570796, 1.971039],accel_mss,speed_ms,0,blend_radius_m)
    movel([0.398416, -1.218288, -2.664127, -0.829974, 1.570796, 1.969213],accel_mss,speed_ms,0,blend_radius_m)
    movel([0.397079, -1.218242, -2.664149, -0.829997, 1.570796, 1.967875],accel_mss,speed_ms,0,blend_radius_m)
    movel([0.396226, -1.217555, -2.664492, -0.830342, 1.570796, 1.967022],accel_mss,speed_ms,0,blend_radius_m)
    movel([0.395959, -1.216391, -2.665070, -0.830928, 1.570796, 1.966756],accel_mss,speed_ms,0,blend_radius_m)
    movel([0.396382, -1.214913, -2.665802, -0.831674, 1.570796, 1.967179],accel_mss,speed_ms,0,blend_radius_m)
    movel([0.397498, -1.213118, -2.666688, -0.832583, 1.570796, 1.968295],accel_mss,speed_ms,0,blend_radius_m)
    movel([0.399310, -1.211002, -2.667728, -0.833659, 1.570796, 1.970106],accel_mss,speed_ms,0,blend_radius_m)
    movel([0.405022, -1.205584, -2.670367, -0.836438, 1.570796, 1.975818],accel_mss,speed_ms,0,blend_radius_m)
    movel([0.413543, -1.198419, -2.673807, -0.840163, 1.570796, 1.984339],accel_mss,speed_ms,0,blend_radius_m)
    movel([0.422369, -1.191559, -2.677048, -0.843782, 1.570796, 1.993165],accel_mss,speed_ms,0,blend_radius_m)
    movel([0.428878, -1.187122, -2.679117, -0.846150, 1.570796, 1.999674],accel_mss,speed_ms,0,blend_radius_m)
    movel([0.431283, -1.185853, -2.679705, -0.846831, 1.570796, 2.002079],accel_mss,speed_ms,0,blend_radius_m)
    movel([0.433167, -1.185257, -2.679980, -0.847152, 1.570796, 2.003963],accel_mss,speed_ms,0,blend_radius_m)
    movel([0.434527, -1.185338, -2.679943, -0.847108, 1.570796, 2.005323],accel_mss,speed_ms,0,blend_radius_m)
    movel([0.435362, -1.186094, -2.679593, -0.846702, 1.570796, 2.006158],accel_mss,speed_ms,0,blend_radius_m)
    movel([0.435577, -1.187342, -2.679015, -0.846032, 1.570796, 2.006373],accel_mss,speed_ms,0,blend_radius_m)
    movel([0.435084, -1.188898, -2.678291, -0.845200, 1.570796, 2.005880],accel_mss,speed_ms,0,blend_radius_m)
    movel([0.433878, -1.190761, -2.677421, -0.844206, 1.570796, 2.004675],accel_mss,speed_ms,0,blend_radius_m)
    movel([0.431974, -1.192924, -2.676407, -0.843058, 1.570796, 2.002770],accel_mss,speed_ms,0,blend_radius_m)
    movel([0.426094, -1.198383, -2.673824, -0.840182, 1.570796, 1.996890],accel_mss,speed_ms,0,blend_radius_m)
    movel([0.417526, -1.205477, -2.670419, -0.836494, 1.570796, 1.988323],accel_mss,speed_ms,0,blend_radius_m)
    speed_ms = 0.003
    movel([0.417526, -1.198293, -2.666816, -0.847281, 1.570796, 1.988323],accel_mss,speed_ms,0,blend_radius_m)
    speed_ms = 0.05
    movel([0.417526, -1.170993, -2.652148, -0.889248, 1.570796, 1.988323],accel_mss,speed_ms,0,blend_radius_m)
    #M_RunCode9
    movel([0.421749, -1.178679, -2.648562, -0.885148, 1.570796, 1.992545],accel_mss,speed_ms,0,blend_radius_m)
    #M_RunCode3
    #num 0 outside
    movel([0.421749, -1.205919, -2.663128, -0.843342, 1.570796, 1.992545],accel_mss,speed_ms,0,blend_radius_m)
    speed_ms = 0.003
    movel([0.421749, -1.213083, -2.666705, -0.832601, 1.570796, 1.992545],accel_mss,speed_ms,0,blend_radius_m)
    speed_ms = 0.015
    movel([0.418589, -1.215448, -2.665537, -0.831403, 1.570796, 1.989385],accel_mss,speed_ms,0,blend_radius_m)
    movel([0.415567, -1.217446, -2.664546, -0.830397, 1.570796, 1.986363],accel_mss,speed_ms,0,blend_radius_m)
    movel([0.412674, -1.219085, -2.663729, -0.829575, 1.570796, 1.983470],accel_mss,speed_ms,0,blend_radius_m)
    movel([0.409911, -1.220363, -2.663090, -0.828936, 1.570796, 1.980707],accel_mss,speed_ms,0,blend_radius_m)
    movel([0.407315, -1.221290, -2.662626, -0.828474, 1.570796, 1.978111],accel_mss,speed_ms,0,blend_radius_m)
    movel([0.404924, -1.221871, -2.662334, -0.828184, 1.570796, 1.975720],accel_mss,speed_ms,0,blend_radius_m)
    movel([0.402734, -1.222111, -2.662214, -0.828065, 1.570796, 1.973530],accel_mss,speed_ms,0,blend_radius_m)
    movel([0.400748, -1.222003, -2.662268, -0.828118, 1.570796, 1.971545],accel_mss,speed_ms,0,blend_radius_m)
    movel([0.398984, -1.221568, -2.662486, -0.828335, 1.570796, 1.969780],accel_mss,speed_ms,0,blend_radius_m)
    movel([0.397463, -1.220832, -2.662856, -0.828702, 1.570796, 1.968260],accel_mss,speed_ms,0,blend_radius_m)
    movel([0.396184, -1.219786, -2.663379, -0.829224, 1.570796, 1.966980],accel_mss,speed_ms,0,blend_radius_m)
    movel([0.395146, -1.218434, -2.664054, -0.829901, 1.570796, 1.965942],accel_mss,speed_ms,0,blend_radius_m)
    movel([0.394396, -1.216841, -2.664847, -0.830701, 1.570796, 1.965192],accel_mss,speed_ms,0,blend_radius_m)
    movel([0.393982, -1.215084, -2.665718, -0.831587, 1.570796, 1.964778],accel_mss,speed_ms,0,blend_radius_m)
    movel([0.393900, -1.213162, -2.666666, -0.832561, 1.570796, 1.964697],accel_mss,speed_ms,0,blend_radius_m)
    movel([0.394161, -1.211065, -2.667697, -0.833627, 1.570796, 1.964958],accel_mss,speed_ms,0,blend_radius_m)
    movel([0.394772, -1.208828, -2.668790, -0.834770, 1.570796, 1.965568],accel_mss,speed_ms,0,blend_radius_m)
    movel([0.395745, -1.206481, -2.669932, -0.835976, 1.570796, 1.966541],accel_mss,speed_ms,0,blend_radius_m)
    movel([0.397083, -1.204017, -2.671124, -0.837248, 1.570796, 1.967879],accel_mss,speed_ms,0,blend_radius_m)
    movel([0.398791, -1.201439, -2.672364, -0.838586, 1.570796, 1.969588],accel_mss,speed_ms,0,blend_radius_m)
    movel([0.400858, -1.198792, -2.673629, -0.839968, 1.570796, 1.971654],accel_mss,speed_ms,0,blend_radius_m)
    movel([0.403274, -1.196129, -2.674894, -0.841365, 1.570796, 1.974071],accel_mss,speed_ms,0,blend_radius_m)
    movel([0.406040, -1.193452, -2.676159, -0.842778, 1.570796, 1.976836],accel_mss,speed_ms,0,blend_radius_m)
    movel([0.409156, -1.190762, -2.677421, -0.844206, 1.570796, 1.979952],accel_mss,speed_ms,0,blend_radius_m)
    movel([0.412397, -1.188248, -2.678594, -0.845547, 1.570796, 1.983193],accel_mss,speed_ms,0,blend_radius_m)
    movel([0.415520, -1.186109, -2.679587, -0.846694, 1.570796, 1.986317],accel_mss,speed_ms,0,blend_radius_m)
    movel([0.418526, -1.184345, -2.680401, -0.847643, 1.570796, 1.989323],accel_mss,speed_ms,0,blend_radius_m)
    movel([0.421407, -1.182966, -2.681036, -0.848387, 1.570796, 1.992203],accel_mss,speed_ms,0,blend_radius_m)
    movel([0.424115, -1.181967, -2.681494, -0.848928, 1.570796, 1.994911],accel_mss,speed_ms,0,blend_radius_m)
    movel([0.426598, -1.181352, -2.681776, -0.849261, 1.570796, 1.997394],accel_mss,speed_ms,0,blend_radius_m)
    movel([0.428858, -1.181116, -2.681884, -0.849389, 1.570796, 1.999654],accel_mss,speed_ms,0,blend_radius_m)
    movel([0.430890, -1.181265, -2.681816, -0.849308, 1.570796, 2.001686],accel_mss,speed_ms,0,blend_radius_m)
    movel([0.432671, -1.181770, -2.681585, -0.849034, 1.570796, 2.003468],accel_mss,speed_ms,0,blend_radius_m)
    movel([0.434190, -1.182603, -2.681203, -0.848584, 1.570796, 2.004986],accel_mss,speed_ms,0,blend_radius_m)
    movel([0.435445, -1.183761, -2.680670, -0.847958, 1.570796, 2.006242],accel_mss,speed_ms,0,blend_radius_m)
    movel([0.436432, -1.185242, -2.679987, -0.847160, 1.570796, 2.007229],accel_mss,speed_ms,0,blend_radius_m)
    movel([0.437113, -1.186965, -2.679190, -0.846234, 1.570796, 2.007909],accel_mss,speed_ms,0,blend_radius_m)
    movel([0.437449, -1.188842, -2.678317, -0.845230, 1.570796, 2.008245],accel_mss,speed_ms,0,blend_radius_m)
    movel([0.437439, -1.190873, -2.677369, -0.844147, 1.570796, 2.008236],accel_mss,speed_ms,0,blend_radius_m)
    movel([0.437088, -1.193056, -2.676345, -0.842988, 1.570796, 2.007885],accel_mss,speed_ms,0,blend_radius_m)
    movel([0.436387, -1.195356, -2.675260, -0.841773, 1.570796, 2.007183],accel_mss,speed_ms,0,blend_radius_m)
    movel([0.435324, -1.197746, -2.674127, -0.840516, 1.570796, 2.006120],accel_mss,speed_ms,0,blend_radius_m)
    movel([0.433899, -1.200225, -2.672945, -0.839219, 1.570796, 2.004695],accel_mss,speed_ms,0,blend_radius_m)
    movel([0.432120, -1.202788, -2.671716, -0.837885, 1.570796, 2.002916],accel_mss,speed_ms,0,blend_radius_m)
    movel([0.430005, -1.205384, -2.670464, -0.836542, 1.570796, 2.000801],accel_mss,speed_ms,0,blend_radius_m)
    movel([0.427569, -1.207965, -2.669211, -0.835213, 1.570796, 1.998365],accel_mss,speed_ms,0,blend_radius_m)
    movel([0.424816, -1.210531, -2.667958, -0.833900, 1.570796, 1.995612],accel_mss,speed_ms,0,blend_radius_m)
    movel([0.421749, -1.213083, -2.666705, -0.832601, 1.570796, 1.992545],accel_mss,speed_ms,0,blend_radius_m)
    speed_ms = 0.003
    movel([0.421749, -1.205919, -2.663128, -0.843342, 1.570796, 1.992545],accel_mss,speed_ms,0,blend_radius_m)
    speed_ms = 0.05
    movel([0.421749, -1.178679, -2.648562, -0.885148, 1.570796, 1.992545],accel_mss,speed_ms,0,blend_radius_m)
    #M_RunCode9
    movel([0.398548, -1.160673, -2.656867, -0.894849, 1.570796, 1.969344],accel_mss,speed_ms,0,blend_radius_m)
    #M_RunCode3
    # num 2
    movel([0.398548, -1.188046, -2.671670, -0.852673, 1.570796, 1.969344],accel_mss,speed_ms,0,blend_radius_m)
    speed_ms = 0.003
    movel([0.398548, -1.195256, -2.675308, -0.841825, 1.570796, 1.969344],accel_mss,speed_ms,0,blend_radius_m)
    speed_ms = 0.02
    movel([0.387519, -1.204390, -2.670944, -0.837055, 1.570796, 1.958316],accel_mss,speed_ms,0,blend_radius_m)
    movel([0.373276, -1.182200, -2.681388, -0.848802, 1.570796, 1.944072],accel_mss,speed_ms,0,blend_radius_m)
    movel([0.374391, -1.181239, -2.681828, -0.849322, 1.570796, 1.945187],accel_mss,speed_ms,0,blend_radius_m)
    movel([0.377402, -1.179045, -2.682829, -0.850514, 1.570796, 1.948199],accel_mss,speed_ms,0,blend_radius_m)
    movel([0.380700, -1.177412, -2.683572, -0.851406, 1.570796, 1.951496],accel_mss,speed_ms,0,blend_radius_m)
    movel([0.384107, -1.176260, -2.684093, -0.852036, 1.570796, 1.954903],accel_mss,speed_ms,0,blend_radius_m)
    movel([0.387437, -1.175507, -2.684433, -0.852448, 1.570796, 1.958233],accel_mss,speed_ms,0,blend_radius_m)
    movel([0.396101, -1.174407, -2.684930, -0.853052, 1.570796, 1.966897],accel_mss,speed_ms,0,blend_radius_m)
    movel([0.404086, -1.173536, -2.685322, -0.853531, 1.570796, 1.974882],accel_mss,speed_ms,0,blend_radius_m)
    movel([0.407182, -1.172914, -2.685601, -0.853874, 1.570796, 1.977978],accel_mss,speed_ms,0,blend_radius_m)
    movel([0.410285, -1.171948, -2.686034, -0.854407, 1.570796, 1.981082],accel_mss,speed_ms,0,blend_radius_m)
    movel([0.413245, -1.170575, -2.686648, -0.855166, 1.570796, 1.984041],accel_mss,speed_ms,0,blend_radius_m)
    movel([0.415914, -1.168726, -2.687472, -0.856191, 1.570796, 1.986710],accel_mss,speed_ms,0,blend_radius_m)
    movel([0.418722, -1.165926, -2.688712, -0.857750, 1.570796, 1.989518],accel_mss,speed_ms,0,blend_radius_m)
    movel([0.419689, -1.164533, -2.689327, -0.858530, 1.570796, 1.990485],accel_mss,speed_ms,0,blend_radius_m)
    movel([0.420364, -1.163144, -2.689937, -0.859308, 1.570796, 1.991160],accel_mss,speed_ms,0,blend_radius_m)
    movel([0.420918, -1.160616, -2.691043, -0.860730, 1.570796, 1.991714],accel_mss,speed_ms,0,blend_radius_m)
    movel([0.420451, -1.158600, -2.691920, -0.861869, 1.570796, 1.991247],accel_mss,speed_ms,0,blend_radius_m)
    movel([0.419659, -1.157633, -2.692340, -0.862417, 1.570796, 1.990456],accel_mss,speed_ms,0,blend_radius_m)
    movel([0.418681, -1.157242, -2.692509, -0.862638, 1.570796, 1.989477],accel_mss,speed_ms,0,blend_radius_m)
    movel([0.417618, -1.157384, -2.692447, -0.862558, 1.570796, 1.988414],accel_mss,speed_ms,0,blend_radius_m)
    movel([0.416582, -1.158002, -2.692180, -0.862208, 1.570796, 1.987378],accel_mss,speed_ms,0,blend_radius_m)
    movel([0.415423, -1.159560, -2.691503, -0.861326, 1.570796, 1.986220],accel_mss,speed_ms,0,blend_radius_m)
    movel([0.414382, -1.161128, -2.690820, -0.860442, 1.570796, 1.985179],accel_mss,speed_ms,0,blend_radius_m)
    movel([0.412740, -1.162760, -2.690106, -0.859524, 1.570796, 1.983536],accel_mss,speed_ms,0,blend_radius_m)
    movel([0.410524, -1.164199, -2.689473, -0.858716, 1.570796, 1.981321],accel_mss,speed_ms,0,blend_radius_m)
    movel([0.408517, -1.164649, -2.689276, -0.858464, 1.570796, 1.979313],accel_mss,speed_ms,0,blend_radius_m)
    movel([0.406864, -1.164233, -2.689459, -0.858697, 1.570796, 1.977661],accel_mss,speed_ms,0,blend_radius_m)
    movel([0.405717, -1.163077, -2.689966, -0.859345, 1.570796, 1.976513],accel_mss,speed_ms,0,blend_radius_m)
    movel([0.405200, -1.161391, -2.690705, -0.860293, 1.570796, 1.975996],accel_mss,speed_ms,0,blend_radius_m)
    movel([0.405438, -1.159373, -2.691584, -0.861432, 1.570796, 1.976234],accel_mss,speed_ms,0,blend_radius_m)
    movel([0.406483, -1.157237, -2.692511, -0.862641, 1.570796, 1.977279],accel_mss,speed_ms,0,blend_radius_m)
    movel([0.408389, -1.155207, -2.693387, -0.863795, 1.570796, 1.979185],accel_mss,speed_ms,0,blend_radius_m)
    movel([0.410308, -1.153825, -2.693981, -0.864583, 1.570796, 1.981104],accel_mss,speed_ms,0,blend_radius_m)
    movel([0.412191, -1.152957, -2.694353, -0.865078, 1.570796, 1.982988],accel_mss,speed_ms,0,blend_radius_m)
    movel([0.414040, -1.152604, -2.694505, -0.865280, 1.570796, 1.984836],accel_mss,speed_ms,0,blend_radius_m)
    movel([0.415848, -1.152773, -2.694432, -0.865184, 1.570796, 1.986644],accel_mss,speed_ms,0,blend_radius_m)
    movel([0.417547, -1.153401, -2.694163, -0.864825, 1.570796, 1.988343],accel_mss,speed_ms,0,blend_radius_m)
    movel([0.419078, -1.154418, -2.693726, -0.864244, 1.570796, 1.989874],accel_mss,speed_ms,0,blend_radius_m)
    movel([0.421621, -1.157629, -2.692341, -0.862419, 1.570796, 1.992417],accel_mss,speed_ms,0,blend_radius_m)
    movel([0.422740, -1.160129, -2.691255, -0.861004, 1.570796, 1.993536],accel_mss,speed_ms,0,blend_radius_m)
    movel([0.423427, -1.162792, -2.690091, -0.859505, 1.570796, 1.994224],accel_mss,speed_ms,0,blend_radius_m)
    movel([0.423686, -1.165609, -2.688852, -0.857927, 1.570796, 1.994483],accel_mss,speed_ms,0,blend_radius_m)
    movel([0.423519, -1.168579, -2.687537, -0.856272, 1.570796, 1.994315],accel_mss,speed_ms,0,blend_radius_m)
    movel([0.422775, -1.171579, -2.686200, -0.854611, 1.570796, 1.993571],accel_mss,speed_ms,0,blend_radius_m)
    movel([0.421289, -1.174496, -2.684890, -0.853003, 1.570796, 1.992085],accel_mss,speed_ms,0,blend_radius_m)
    movel([0.419070, -1.177328, -2.683609, -0.851451, 1.570796, 1.989866],accel_mss,speed_ms,0,blend_radius_m)
    movel([0.416125, -1.180080, -2.682358, -0.849952, 1.570796, 1.986922],accel_mss,speed_ms,0,blend_radius_m)
    movel([0.413191, -1.182183, -2.681395, -0.848811, 1.570796, 1.983988],accel_mss,speed_ms,0,blend_radius_m)
    movel([0.410228, -1.183711, -2.680693, -0.847984, 1.570796, 1.981024],accel_mss,speed_ms,0,blend_radius_m)
    movel([0.407305, -1.184765, -2.680207, -0.847416, 1.570796, 1.978101],accel_mss,speed_ms,0,blend_radius_m)
    movel([0.404499, -1.185444, -2.679894, -0.847051, 1.570796, 1.975295],accel_mss,speed_ms,0,blend_radius_m)
    movel([0.397845, -1.186264, -2.679515, -0.846611, 1.570796, 1.968641],accel_mss,speed_ms,0,blend_radius_m)
    movel([0.391540, -1.187111, -2.679122, -0.846156, 1.570796, 1.962337],accel_mss,speed_ms,0,blend_radius_m)
    movel([0.388986, -1.187747, -2.678827, -0.845815, 1.570796, 1.959782],accel_mss,speed_ms,0,blend_radius_m)
    movel([0.386370, -1.188709, -2.678379, -0.845301, 1.570796, 1.957167],accel_mss,speed_ms,0,blend_radius_m)
    movel([0.383776, -1.190069, -2.677745, -0.844575, 1.570796, 1.954572],accel_mss,speed_ms,0,blend_radius_m)
    movel([0.381297, -1.191889, -2.676893, -0.843607, 1.570796, 1.952094],accel_mss,speed_ms,0,blend_radius_m)
    movel([0.381830, -1.192722, -2.676502, -0.843165, 1.570796, 1.952626],accel_mss,speed_ms,0,blend_radius_m)
    movel([0.383468, -1.194889, -2.675481, -0.842019, 1.570796, 1.954264],accel_mss,speed_ms,0,blend_radius_m)
    movel([0.385262, -1.196485, -2.674726, -0.841178, 1.570796, 1.956059],accel_mss,speed_ms,0,blend_radius_m)
    movel([0.387208, -1.197517, -2.674236, -0.840636, 1.570796, 1.958005],accel_mss,speed_ms,0,blend_radius_m)
    movel([0.389316, -1.197985, -2.674013, -0.840391, 1.570796, 1.960112],accel_mss,speed_ms,0,blend_radius_m)
    movel([0.391528, -1.197956, -2.674027, -0.840406, 1.570796, 1.962325],accel_mss,speed_ms,0,blend_radius_m)
    movel([0.393803, -1.197493, -2.674247, -0.840649, 1.570796, 1.964599],accel_mss,speed_ms,0,blend_radius_m)
    movel([0.396140, -1.196594, -2.674674, -0.841121, 1.570796, 1.966936],accel_mss,speed_ms,0,blend_radius_m)
    movel([0.398548, -1.195256, -2.675308, -0.841825, 1.570796, 1.969344],accel_mss,speed_ms,0,blend_radius_m)
    speed_ms = 0.003
    movel([0.398548, -1.188046, -2.671670, -0.852673, 1.570796, 1.969344],accel_mss,speed_ms,0,blend_radius_m)
    speed_ms = 0.05
    movel([0.398548, -1.160673, -2.656867, -0.894849, 1.570796, 1.969344],accel_mss,speed_ms,0,blend_radius_m)
    #M_RunCode9
    movel([0.492183, -1.374535, -2.534046, -0.803807, 1.570796, 2.062980],accel_mss,speed_ms,0,blend_radius_m)
    #M_RunCode3
    movel([0.492183, -1.399008, -2.546063, -0.767317, 1.570796, 2.062980],accel_mss,speed_ms,0,blend_radius_m)
    speed_ms = 0.003
    movel([0.492183, -1.405355, -2.548996, -0.758039, 1.570796, 2.062980],accel_mss,speed_ms,0,blend_radius_m)
    speed_ms = 0.02
    movel([0.494554, -1.404214, -2.549842, -0.758333, 1.570796, 2.065351],accel_mss,speed_ms,0,blend_radius_m)
    movel([0.497069, -1.403547, -2.550337, -0.758505, 1.570796, 2.067866],accel_mss,speed_ms,0,blend_radius_m)
    movel([0.499611, -1.403261, -2.550549, -0.758580, 1.570796, 2.070408],accel_mss,speed_ms,0,blend_radius_m)
    movel([0.502055, -1.403267, -2.550544, -0.758578, 1.570796, 2.072851],accel_mss,speed_ms,0,blend_radius_m)
    movel([0.508325, -1.403916, -2.550063, -0.758410, 1.570796, 2.079121],accel_mss,speed_ms,0,blend_radius_m)
    movel([0.514086, -1.404611, -2.549548, -0.758230, 1.570796, 2.084883],accel_mss,speed_ms,0,blend_radius_m)
    movel([0.516344, -1.404668, -2.549506, -0.758215, 1.570796, 2.087141],accel_mss,speed_ms,0,blend_radius_m)
    movel([0.518640, -1.404466, -2.549656, -0.758268, 1.570796, 2.089437],accel_mss,speed_ms,0,blend_radius_m)
    movel([0.520871, -1.403935, -2.550049, -0.758405, 1.570796, 2.091667],accel_mss,speed_ms,0,blend_radius_m)
    movel([0.522937, -1.403002, -2.550740, -0.758647, 1.570796, 2.093733],accel_mss,speed_ms,0,blend_radius_m)
    movel([0.525186, -1.401385, -2.551934, -0.759070, 1.570796, 2.095982],accel_mss,speed_ms,0,blend_radius_m)
    movel([0.525999, -1.400510, -2.552579, -0.759300, 1.570796, 2.096795],accel_mss,speed_ms,0,blend_radius_m)
    movel([0.526604, -1.399591, -2.553255, -0.759543, 1.570796, 2.097401],accel_mss,speed_ms,0,blend_radius_m)
    movel([0.527228, -1.397806, -2.554564, -0.760019, 1.570796, 2.098024],accel_mss,speed_ms,0,blend_radius_m)
    movel([0.527082, -1.396230, -2.555715, -0.760443, 1.570796, 2.097878],accel_mss,speed_ms,0,blend_radius_m)
    movel([0.526613, -1.395377, -2.556338, -0.760674, 1.570796, 2.097409],accel_mss,speed_ms,0,blend_radius_m)
    movel([0.525954, -1.394923, -2.556668, -0.760798, 1.570796, 2.096751],accel_mss,speed_ms,0,blend_radius_m)
    movel([0.525193, -1.394847, -2.556724, -0.760818, 1.570796, 2.095990],accel_mss,speed_ms,0,blend_radius_m)
    movel([0.524404, -1.395130, -2.556518, -0.760741, 1.570796, 2.095201],accel_mss,speed_ms,0,blend_radius_m)
    movel([0.523441, -1.396092, -2.555816, -0.760481, 1.570796, 2.094237],accel_mss,speed_ms,0,blend_radius_m)
    movel([0.522557, -1.397084, -2.555092, -0.760213, 1.570796, 2.093354],accel_mss,speed_ms,0,blend_radius_m)
    movel([0.521242, -1.398019, -2.554408, -0.759962, 1.570796, 2.092038],accel_mss,speed_ms,0,blend_radius_m)
    movel([0.519539, -1.398719, -2.553894, -0.759775, 1.570796, 2.090335],accel_mss,speed_ms,0,blend_radius_m)
    movel([0.518076, -1.398712, -2.553900, -0.759777, 1.570796, 2.088872],accel_mss,speed_ms,0,blend_radius_m)
    movel([0.516943, -1.398121, -2.554333, -0.759935, 1.570796, 2.087739],accel_mss,speed_ms,0,blend_radius_m)
    movel([0.516241, -1.397065, -2.555106, -0.760218, 1.570796, 2.087037],accel_mss,speed_ms,0,blend_radius_m)
    movel([0.516038, -1.395715, -2.556091, -0.760583, 1.570796, 2.086834],accel_mss,speed_ms,0,blend_radius_m)
    movel([0.516399, -1.394250, -2.557158, -0.760981, 1.570796, 2.087195],accel_mss,speed_ms,0,blend_radius_m)
    movel([0.517341, -1.392838, -2.558183, -0.761368, 1.570796, 2.088137],accel_mss,speed_ms,0,blend_radius_m)
    movel([0.518880, -1.391654, -2.559040, -0.761695, 1.570796, 2.089676],accel_mss,speed_ms,0,blend_radius_m)
    movel([0.520364, -1.390953, -2.559547, -0.761889, 1.570796, 2.091161],accel_mss,speed_ms,0,blend_radius_m)
    movel([0.521777, -1.390632, -2.559779, -0.761979, 1.570796, 2.092573],accel_mss,speed_ms,0,blend_radius_m)
    movel([0.523112, -1.390689, -2.559738, -0.761963, 1.570796, 2.093908],accel_mss,speed_ms,0,blend_radius_m)
    movel([0.524369, -1.391124, -2.559423, -0.761842, 1.570796, 2.095165],accel_mss,speed_ms,0,blend_radius_m)
    movel([0.525510, -1.391878, -2.558878, -0.761633, 1.570796, 2.096306],accel_mss,speed_ms,0,blend_radius_m)
    movel([0.526495, -1.392895, -2.558141, -0.761352, 1.570796, 2.097291],accel_mss,speed_ms,0,blend_radius_m)
    movel([0.527999, -1.395705, -2.556099, -0.760585, 1.570796, 2.098795],accel_mss,speed_ms,0,blend_radius_m)
    movel([0.528561, -1.397751, -2.554604, -0.760034, 1.570796, 2.099357],accel_mss,speed_ms,0,blend_radius_m)
    movel([0.528805, -1.399842, -2.553070, -0.759477, 1.570796, 2.099602],accel_mss,speed_ms,0,blend_radius_m)
    movel([0.528733, -1.401977, -2.551497, -0.758914, 1.570796, 2.099529],accel_mss,speed_ms,0,blend_radius_m)
    movel([0.528346, -1.404157, -2.549884, -0.758347, 1.570796, 2.099142],accel_mss,speed_ms,0,blend_radius_m)
    movel([0.527544, -1.406266, -2.548318, -0.757805, 1.570796, 2.098340],accel_mss,speed_ms,0,blend_radius_m)
    movel([0.526223, -1.408195, -2.546879, -0.757315, 1.570796, 2.097019],accel_mss,speed_ms,0,blend_radius_m)
    movel([0.524388, -1.409944, -2.545570, -0.756875, 1.570796, 2.095185],accel_mss,speed_ms,0,blend_radius_m)
    movel([0.522037, -1.411516, -2.544389, -0.756484, 1.570796, 2.092833],accel_mss,speed_ms,0,blend_radius_m)
    movel([0.519753, -1.412609, -2.543566, -0.756214, 1.570796, 2.090549],accel_mss,speed_ms,0,blend_radius_m)
    movel([0.517497, -1.413267, -2.543069, -0.756052, 1.570796, 2.088293],accel_mss,speed_ms,0,blend_radius_m)
    movel([0.515310, -1.413576, -2.542836, -0.755977, 1.570796, 2.086106],accel_mss,speed_ms,0,blend_radius_m)
    movel([0.513244, -1.413623, -2.542801, -0.755965, 1.570796, 2.084041],accel_mss,speed_ms,0,blend_radius_m)
    movel([0.508414, -1.413136, -2.543169, -0.756085, 1.570796, 2.079211],accel_mss,speed_ms,0,blend_radius_m)
    movel([0.503828, -1.412721, -2.543481, -0.756187, 1.570796, 2.074625],accel_mss,speed_ms,0,blend_radius_m)
    movel([0.501942, -1.412771, -2.543444, -0.756174, 1.570796, 2.072738],accel_mss,speed_ms,0,blend_radius_m)
    movel([0.499976, -1.413061, -2.543225, -0.756103, 1.570796, 2.070772],accel_mss,speed_ms,0,blend_radius_m)
    movel([0.497984, -1.413655, -2.542777, -0.755957, 1.570796, 2.068780],accel_mss,speed_ms,0,blend_radius_m)
    movel([0.496027, -1.414618, -2.542049, -0.755723, 1.570796, 2.066824],accel_mss,speed_ms,0,blend_radius_m)
    movel([0.496323, -1.415340, -2.541501, -0.755547, 1.570796, 2.067119],accel_mss,speed_ms,0,blend_radius_m)
    movel([0.497281, -1.417258, -2.540045, -0.755086, 1.570796, 2.068077],accel_mss,speed_ms,0,blend_radius_m)
    movel([0.498406, -1.418772, -2.538892, -0.754725, 1.570796, 2.069203],accel_mss,speed_ms,0,blend_radius_m)
    movel([0.499699, -1.419880, -2.538046, -0.754464, 1.570796, 2.070495],accel_mss,speed_ms,0,blend_radius_m)
    movel([0.501162, -1.420584, -2.537507, -0.754298, 1.570796, 2.071959],accel_mss,speed_ms,0,blend_radius_m)
    movel([0.502754, -1.420928, -2.537243, -0.754218, 1.570796, 2.073551],accel_mss,speed_ms,0,blend_radius_m)
    movel([0.504429, -1.420952, -2.537225, -0.754212, 1.570796, 2.075225],accel_mss,speed_ms,0,blend_radius_m)
    movel([0.506194, -1.420656, -2.537451, -0.754281, 1.570796, 2.076990],accel_mss,speed_ms,0,blend_radius_m)
    movel([0.508047, -1.420040, -2.537923, -0.754426, 1.570796, 2.078844],accel_mss,speed_ms,0,blend_radius_m)
    movel([0.499242, -1.425154, -2.533992, -0.753243, 1.570796, 2.070038],accel_mss,speed_ms,0,blend_radius_m)
    movel([0.491288, -1.405893, -2.548595, -0.757901, 1.570796, 2.062085],accel_mss,speed_ms,0,blend_radius_m)
    movel([0.492183, -1.405355, -2.548996, -0.758039, 1.570796, 2.062980],accel_mss,speed_ms,0,blend_radius_m)
    speed_ms = 0.003
    movel([0.492183, -1.399008, -2.546063, -0.767317, 1.570796, 2.062980],accel_mss,speed_ms,0,blend_radius_m)
    speed_ms = 0.05
    movel([0.492183, -1.374535, -2.534046, -0.803807, 1.570796, 2.062980],accel_mss,speed_ms,0,blend_radius_m)
    #M_RunCode9
    movel([0.505685, -1.394015, -2.519960, -0.798414, 1.570796, 2.076481],accel_mss,speed_ms,0,blend_radius_m)
    #M_RunCode3
    movel([0.505685, -1.418115, -2.531735, -0.762539, 1.570796, 2.076481],accel_mss,speed_ms,0,blend_radius_m)
    speed_ms = 0.003
    movel([0.505685, -1.424358, -2.534606, -0.753424, 1.570796, 2.076481],accel_mss,speed_ms,0,blend_radius_m)
    speed_ms = 0.02
    movel([0.507343, -1.423678, -2.535131, -0.753580, 1.570796, 2.078139],accel_mss,speed_ms,0,blend_radius_m)
    movel([0.508789, -1.423672, -2.535136, -0.753582, 1.570796, 2.079585],accel_mss,speed_ms,0,blend_radius_m)
    movel([0.509918, -1.424231, -2.534705, -0.753454, 1.570796, 2.080714],accel_mss,speed_ms,0,blend_radius_m)
    movel([0.510614, -1.425248, -2.533920, -0.753222, 1.570796, 2.081410],accel_mss,speed_ms,0,blend_radius_m)
    movel([0.510814, -1.426544, -2.532917, -0.752928, 1.570796, 2.081610],accel_mss,speed_ms,0,blend_radius_m)
    movel([0.510452, -1.427953, -2.531824, -0.752612, 1.570796, 2.081249],accel_mss,speed_ms,0,blend_radius_m)
    movel([0.509538, -1.429300, -2.530776, -0.752313, 1.570796, 2.080334],accel_mss,speed_ms,0,blend_radius_m)
    movel([0.508067, -1.430415, -2.529908, -0.752067, 1.570796, 2.078864],accel_mss,speed_ms,0,blend_radius_m)
    movel([0.506703, -1.431026, -2.529430, -0.751933, 1.570796, 2.077499],accel_mss,speed_ms,0,blend_radius_m)
    movel([0.505574, -1.431213, -2.529284, -0.751892, 1.570796, 2.076370],accel_mss,speed_ms,0,blend_radius_m)
    movel([0.504412, -1.431493, -2.529065, -0.751831, 1.570796, 2.075208],accel_mss,speed_ms,0,blend_radius_m)
    movel([0.503766, -1.432035, -2.528641, -0.751713, 1.570796, 2.074562],accel_mss,speed_ms,0,blend_radius_m)
    movel([0.503353, -1.432783, -2.528055, -0.751551, 1.570796, 2.074150],accel_mss,speed_ms,0,blend_radius_m)
    movel([0.503206, -1.433607, -2.527409, -0.751373, 1.570796, 2.074002],accel_mss,speed_ms,0,blend_radius_m)
    movel([0.503356, -1.434381, -2.526800, -0.751208, 1.570796, 2.074152],accel_mss,speed_ms,0,blend_radius_m)
    movel([0.503856, -1.435229, -2.526133, -0.751027, 1.570796, 2.074653],accel_mss,speed_ms,0,blend_radius_m)
    movel([0.504583, -1.435849, -2.525645, -0.750896, 1.570796, 2.075379],accel_mss,speed_ms,0,blend_radius_m)
    movel([0.505535, -1.436238, -2.525338, -0.750814, 1.570796, 2.076331],accel_mss,speed_ms,0,blend_radius_m)
    movel([0.506718, -1.436396, -2.525213, -0.750780, 1.570796, 2.077514],accel_mss,speed_ms,0,blend_radius_m)
    movel([0.508056, -1.436320, -2.525273, -0.750796, 1.570796, 2.078852],accel_mss,speed_ms,0,blend_radius_m)
    movel([0.509486, -1.435996, -2.525528, -0.750865, 1.570796, 2.080282],accel_mss,speed_ms,0,blend_radius_m)
    movel([0.511004, -1.435426, -2.525978, -0.750985, 1.570796, 2.081801],accel_mss,speed_ms,0,blend_radius_m)
    movel([0.512618, -1.434610, -2.526620, -0.751159, 1.570796, 2.083414],accel_mss,speed_ms,0,blend_radius_m)
    movel([0.515148, -1.432826, -2.528022, -0.751542, 1.570796, 2.085945],accel_mss,speed_ms,0,blend_radius_m)
    movel([0.517198, -1.430614, -2.529752, -0.752023, 1.570796, 2.087995],accel_mss,speed_ms,0,blend_radius_m)
    movel([0.518018, -1.429355, -2.530734, -0.752300, 1.570796, 2.088814],accel_mss,speed_ms,0,blend_radius_m)
    movel([0.518663, -1.428007, -2.531782, -0.752600, 1.570796, 2.089459],accel_mss,speed_ms,0,blend_radius_m)
    movel([0.519439, -1.425040, -2.534080, -0.753269, 1.570796, 2.090235],accel_mss,speed_ms,0,blend_radius_m)
    movel([0.519436, -1.421793, -2.536580, -0.754016, 1.570796, 2.090232],accel_mss,speed_ms,0,blend_radius_m)
    movel([0.518555, -1.418352, -2.539212, -0.754825, 1.570796, 2.089351],accel_mss,speed_ms,0,blend_radius_m)
    movel([0.532257, -1.410606, -2.545073, -0.756710, 1.570796, 2.103054],accel_mss,speed_ms,0,blend_radius_m)
    movel([0.537415, -1.425473, -2.533745, -0.753170, 1.570796, 2.108212],accel_mss,speed_ms,0,blend_radius_m)
    movel([0.528594, -1.430343, -2.529963, -0.752083, 1.570796, 2.099390],accel_mss,speed_ms,0,blend_radius_m)
    movel([0.530498, -1.428621, -2.531305, -0.752463, 1.570796, 2.101294],accel_mss,speed_ms,0,blend_radius_m)
    movel([0.532054, -1.426533, -2.532925, -0.752931, 1.570796, 2.102850],accel_mss,speed_ms,0,blend_radius_m)
    movel([0.533176, -1.424184, -2.534740, -0.753464, 1.570796, 2.103972],accel_mss,speed_ms,0,blend_radius_m)
    movel([0.533790, -1.421674, -2.536671, -0.754044, 1.570796, 2.104586],accel_mss,speed_ms,0,blend_radius_m)
    movel([0.533838, -1.419100, -2.538642, -0.754648, 1.570796, 2.104634],accel_mss,speed_ms,0,blend_radius_m)
    movel([0.533270, -1.416566, -2.540572, -0.755252, 1.570796, 2.104066],accel_mss,speed_ms,0,blend_radius_m)
    movel([0.523200, -1.422207, -2.536262, -0.753920, 1.570796, 2.093996],accel_mss,speed_ms,0,blend_radius_m)
    movel([0.523982, -1.425264, -2.533907, -0.753218, 1.570796, 2.094778],accel_mss,speed_ms,0,blend_radius_m)
    movel([0.524165, -1.428496, -2.531402, -0.752491, 1.570796, 2.094961],accel_mss,speed_ms,0,blend_radius_m)
    movel([0.523653, -1.431730, -2.528880, -0.751779, 1.570796, 2.094449],accel_mss,speed_ms,0,blend_radius_m)
    movel([0.523103, -1.433286, -2.527660, -0.751442, 1.570796, 2.093899],accel_mss,speed_ms,0,blend_radius_m)
    movel([0.522353, -1.434804, -2.526468, -0.751117, 1.570796, 2.093149],accel_mss,speed_ms,0,blend_radius_m)
    movel([0.521392, -1.436236, -2.525339, -0.750814, 1.570796, 2.092189],accel_mss,speed_ms,0,blend_radius_m)
    movel([0.520203, -1.437537, -2.524311, -0.750541, 1.570796, 2.090999],accel_mss,speed_ms,0,blend_radius_m)
    movel([0.518786, -1.438713, -2.523380, -0.750296, 1.570796, 2.089582],accel_mss,speed_ms,0,blend_radius_m)
    movel([0.517140, -1.439760, -2.522548, -0.750080, 1.570796, 2.087936],accel_mss,speed_ms,0,blend_radius_m)
    movel([0.515419, -1.440606, -2.521876, -0.749907, 1.570796, 2.086215],accel_mss,speed_ms,0,blend_radius_m)
    movel([0.513770, -1.441178, -2.521420, -0.749790, 1.570796, 2.084567],accel_mss,speed_ms,0,blend_radius_m)
    movel([0.512194, -1.441476, -2.521183, -0.749730, 1.570796, 2.082991],accel_mss,speed_ms,0,blend_radius_m)
    movel([0.510687, -1.441499, -2.521165, -0.749725, 1.570796, 2.081483],accel_mss,speed_ms,0,blend_radius_m)
    movel([0.507968, -1.440895, -2.521646, -0.749848, 1.570796, 2.078764],accel_mss,speed_ms,0,blend_radius_m)
    movel([0.505701, -1.439532, -2.522730, -0.750127, 1.570796, 2.076497],accel_mss,speed_ms,0,blend_radius_m)
    movel([0.503914, -1.437597, -2.524264, -0.750528, 1.570796, 2.074711],accel_mss,speed_ms,0,blend_radius_m)
    movel([0.502646, -1.435274, -2.526097, -0.751017, 1.570796, 2.073442],accel_mss,speed_ms,0,blend_radius_m)
    movel([0.502142, -1.433468, -2.527518, -0.751403, 1.570796, 2.072938],accel_mss,speed_ms,0,blend_radius_m)
    movel([0.501979, -1.431437, -2.529109, -0.751843, 1.570796, 2.072776],accel_mss,speed_ms,0,blend_radius_m)
    movel([0.502213, -1.429345, -2.530741, -0.752303, 1.570796, 2.073009],accel_mss,speed_ms,0,blend_radius_m)
    movel([0.502903, -1.427364, -2.532281, -0.752744, 1.570796, 2.073699],accel_mss,speed_ms,0,blend_radius_m)
    movel([0.504056, -1.425650, -2.533608, -0.753130, 1.570796, 2.074852],accel_mss,speed_ms,0,blend_radius_m)
    movel([0.505685, -1.424358, -2.534606, -0.753424, 1.570796, 2.076481],accel_mss,speed_ms,0,blend_radius_m)
    speed_ms = 0.003
    movel([0.505685, -1.418115, -2.531735, -0.762539, 1.570796, 2.076481],accel_mss,speed_ms,0,blend_radius_m)
    speed_ms = 0.05
    movel([0.505685, -1.394015, -2.519960, -0.798414, 1.570796, 2.076481],accel_mss,speed_ms,0,blend_radius_m)
    #M_RunCode9
    movel([0.511765, -1.313908, -2.574588, -0.823893, 1.570796, 2.082561],accel_mss,speed_ms,0,blend_radius_m)
    #M_RunCode3
    movel([0.511765, -1.339451, -2.587378, -0.785560, 1.570796, 2.082561],accel_mss,speed_ms,0,blend_radius_m)
    speed_ms = 0.003
    movel([0.511765, -1.346101, -2.590505, -0.775783, 1.570796, 2.082561],accel_mss,speed_ms,0,blend_radius_m)
    speed_ms = 0.02
    movel([0.509003, -1.346634, -2.590154, -0.775602, 1.570796, 2.079799],accel_mss,speed_ms,0,blend_radius_m)
    movel([0.506323, -1.346604, -2.590173, -0.775612, 1.570796, 2.077120],accel_mss,speed_ms,0,blend_radius_m)
    movel([0.503779, -1.346109, -2.590499, -0.775781, 1.570796, 2.074576],accel_mss,speed_ms,0,blend_radius_m)
    movel([0.501429, -1.345241, -2.591071, -0.776077, 1.570796, 2.072225],accel_mss,speed_ms,0,blend_radius_m)
    movel([0.499334, -1.344090, -2.591827, -0.776472, 1.570796, 2.070130],accel_mss,speed_ms,0,blend_radius_m)
    movel([0.500903, -1.340898, -2.593914, -0.777577, 1.570796, 2.071699],accel_mss,speed_ms,0,blend_radius_m)
    movel([0.503381, -1.337486, -2.596130, -0.778773, 1.570796, 2.074177],accel_mss,speed_ms,0,blend_radius_m)
    movel([0.506519, -1.334154, -2.598278, -0.779957, 1.570796, 2.077315],accel_mss,speed_ms,0,blend_radius_m)
    movel([0.510041, -1.331225, -2.600155, -0.781010, 1.570796, 2.080838],accel_mss,speed_ms,0,blend_radius_m)
    movel([0.513677, -1.329019, -2.601560, -0.781810, 1.570796, 2.084474],accel_mss,speed_ms,0,blend_radius_m)
    movel([0.515448, -1.328288, -2.602024, -0.782077, 1.570796, 2.086244],accel_mss,speed_ms,0,blend_radius_m)
    movel([0.517140, -1.327859, -2.602297, -0.782234, 1.570796, 2.087936],accel_mss,speed_ms,0,blend_radius_m)
    movel([0.518717, -1.327772, -2.602352, -0.782265, 1.570796, 2.089514],accel_mss,speed_ms,0,blend_radius_m)
    movel([0.520146, -1.328066, -2.602165, -0.782158, 1.570796, 2.090942],accel_mss,speed_ms,0,blend_radius_m)
    movel([0.521388, -1.328777, -2.601714, -0.781898, 1.570796, 2.092184],accel_mss,speed_ms,0,blend_radius_m)
    movel([0.522405, -1.329948, -2.600969, -0.781472, 1.570796, 2.093201],accel_mss,speed_ms,0,blend_radius_m)
    movel([0.523173, -1.332184, -2.599542, -0.780663, 1.570796, 2.093970],accel_mss,speed_ms,0,blend_radius_m)
    movel([0.522946, -1.334699, -2.597928, -0.779762, 1.570796, 2.093742],accel_mss,speed_ms,0,blend_radius_m)
    movel([0.521842, -1.337390, -2.596192, -0.778807, 1.570796, 2.092638],accel_mss,speed_ms,0,blend_radius_m)
    movel([0.519982, -1.340150, -2.594401, -0.777838, 1.570796, 2.090778],accel_mss,speed_ms,0,blend_radius_m)
    movel([0.517307, -1.342963, -2.592565, -0.776861, 1.570796, 2.088104],accel_mss,speed_ms,0,blend_radius_m)
    movel([0.514551, -1.344910, -2.591288, -0.776190, 1.570796, 2.085348],accel_mss,speed_ms,0,blend_radius_m)
    movel([0.511765, -1.346101, -2.590505, -0.775783, 1.570796, 2.082561],accel_mss,speed_ms,0,blend_radius_m)
    speed_ms = 0.003
    movel([0.511765, -1.339451, -2.587378, -0.785560, 1.570796, 2.082561],accel_mss,speed_ms,0,blend_radius_m)
    speed_ms = 0.05
    movel([0.511765, -1.313908, -2.574588, -0.823893, 1.570796, 2.082561],accel_mss,speed_ms,0,blend_radius_m)
    #M_RunCode9
    movel([0.593175, -1.228303, -2.623878, -0.860208, 1.570796, 2.163971],accel_mss,speed_ms,0,blend_radius_m)
    #M_RunCode3
    movel([0.593175, -1.255054, -2.637790, -0.819545, 1.570796, 2.163971],accel_mss,speed_ms,0,blend_radius_m)
    speed_ms = 0.003
    movel([0.593175, -1.262061, -2.641200, -0.809128, 1.570796, 2.163971],accel_mss,speed_ms,0,blend_radius_m)
    speed_ms = 0.02
    movel([0.592118, -1.260949, -2.641811, -0.809629, 1.570796, 2.162914],accel_mss,speed_ms,0,blend_radius_m)
    movel([0.591505, -1.259430, -2.642643, -0.810317, 1.570796, 2.162302],accel_mss,speed_ms,0,blend_radius_m)
    movel([0.591148, -1.257700, -2.643586, -0.811103, 1.570796, 2.161944],accel_mss,speed_ms,0,blend_radius_m)
    movel([0.591952, -1.257478, -2.643707, -0.811204, 1.570796, 2.162749],accel_mss,speed_ms,0,blend_radius_m)
    movel([0.592411, -1.257816, -2.643523, -0.811050, 1.570796, 2.163207],accel_mss,speed_ms,0,blend_radius_m)
    movel([0.592987, -1.258156, -2.643338, -0.810895, 1.570796, 2.163783],accel_mss,speed_ms,0,blend_radius_m)
    movel([0.594138, -1.257945, -2.643453, -0.810991, 1.570796, 2.164934],accel_mss,speed_ms,0,blend_radius_m)
    movel([0.595427, -1.257217, -2.643850, -0.811323, 1.570796, 2.166224],accel_mss,speed_ms,0,blend_radius_m)
    movel([0.596669, -1.256262, -2.644368, -0.811759, 1.570796, 2.167466],accel_mss,speed_ms,0,blend_radius_m)
    movel([0.598371, -1.254882, -2.645116, -0.812391, 1.570796, 2.169167],accel_mss,speed_ms,0,blend_radius_m)
    movel([0.598070, -1.252620, -2.646337, -0.813432, 1.570796, 2.168867],accel_mss,speed_ms,0,blend_radius_m)
    movel([0.597149, -1.251145, -2.647130, -0.814114, 1.570796, 2.167945],accel_mss,speed_ms,0,blend_radius_m)
    movel([0.596399, -1.250811, -2.647309, -0.814269, 1.570796, 2.167195],accel_mss,speed_ms,0,blend_radius_m)
    movel([0.595425, -1.250808, -2.647311, -0.814270, 1.570796, 2.166221],accel_mss,speed_ms,0,blend_radius_m)
    movel([0.594204, -1.251181, -2.647110, -0.814097, 1.570796, 2.165000],accel_mss,speed_ms,0,blend_radius_m)
    movel([0.592717, -1.251976, -2.646684, -0.813730, 1.570796, 2.163513],accel_mss,speed_ms,0,blend_radius_m)
    movel([0.593308, -1.250419, -2.647519, -0.814451, 1.570796, 2.164105],accel_mss,speed_ms,0,blend_radius_m)
    movel([0.593995, -1.249081, -2.648235, -0.815073, 1.570796, 2.164792],accel_mss,speed_ms,0,blend_radius_m)
    movel([0.594412, -1.248607, -2.648488, -0.815294, 1.570796, 2.165208],accel_mss,speed_ms,0,blend_radius_m)
    movel([0.594899, -1.248328, -2.648637, -0.815424, 1.570796, 2.165695],accel_mss,speed_ms,0,blend_radius_m)
    movel([0.596139, -1.248534, -2.648527, -0.815328, 1.570796, 2.166935],accel_mss,speed_ms,0,blend_radius_m)
    movel([0.597985, -1.249993, -2.647747, -0.814649, 1.570796, 2.168781],accel_mss,speed_ms,0,blend_radius_m)
    movel([0.599239, -1.252067, -2.646635, -0.813688, 1.570796, 2.170035],accel_mss,speed_ms,0,blend_radius_m)
    movel([0.599500, -1.253288, -2.645977, -0.813124, 1.570796, 2.170297],accel_mss,speed_ms,0,blend_radius_m)
    movel([0.599438, -1.254612, -2.645262, -0.812515, 1.570796, 2.170234],accel_mss,speed_ms,0,blend_radius_m)
    movel([0.598999, -1.256018, -2.644501, -0.811870, 1.570796, 2.169795],accel_mss,speed_ms,0,blend_radius_m)
    movel([0.598125, -1.257489, -2.643701, -0.811199, 1.570796, 2.168921],accel_mss,speed_ms,0,blend_radius_m)
    movel([0.596913, -1.256631, -2.644168, -0.811590, 1.570796, 2.167709],accel_mss,speed_ms,0,blend_radius_m)
    movel([0.594869, -1.262559, -2.640926, -0.808904, 1.570796, 2.165665],accel_mss,speed_ms,0,blend_radius_m)
    movel([0.593175, -1.262061, -2.641200, -0.809128, 1.570796, 2.163971],accel_mss,speed_ms,0,blend_radius_m)
    speed_ms = 0.003
    movel([0.593175, -1.255054, -2.637790, -0.819545, 1.570796, 2.163971],accel_mss,speed_ms,0,blend_radius_m)
    speed_ms = 0.05
    movel([0.593175, -1.228303, -2.623878, -0.860208, 1.570796, 2.163971],accel_mss,speed_ms,0,blend_radius_m)
    #M_RunCode9
    movel([0.574585, -1.187672, -2.644287, -0.880430, 1.570796, 2.145381],accel_mss,speed_ms,0,blend_radius_m)
    #M_RunCode3
    movel([0.574585, -1.214836, -2.658735, -0.838818, 1.570796, 2.145381],accel_mss,speed_ms,0,blend_radius_m)
    speed_ms = 0.003
    movel([0.574585, -1.221975, -2.662282, -0.828132, 1.570796, 2.145381],accel_mss,speed_ms,0,blend_radius_m)
    speed_ms = 0.02
    movel([0.571968, -1.223903, -2.661311, -0.827175, 1.570796, 2.142764],accel_mss,speed_ms,0,blend_radius_m)
    movel([0.569236, -1.225606, -2.660449, -0.826333, 1.570796, 2.140032],accel_mss,speed_ms,0,blend_radius_m)
    movel([0.566418, -1.227048, -2.659718, -0.825623, 1.570796, 2.137214],accel_mss,speed_ms,0,blend_radius_m)
    movel([0.563541, -1.228201, -2.659131, -0.825057, 1.570796, 2.134337],accel_mss,speed_ms,0,blend_radius_m)
    movel([0.560640, -1.229035, -2.658705, -0.824649, 1.570796, 2.131436],accel_mss,speed_ms,0,blend_radius_m)
    movel([0.559180, -1.229158, -2.658643, -0.824589, 1.570796, 2.129976],accel_mss,speed_ms,0,blend_radius_m)
    movel([0.557735, -1.229044, -2.658701, -0.824644, 1.570796, 2.128531],accel_mss,speed_ms,0,blend_radius_m)
    movel([0.556429, -1.228954, -2.658747, -0.824688, 1.570796, 2.127225],accel_mss,speed_ms,0,blend_radius_m)
    movel([0.555404, -1.229136, -2.658654, -0.824599, 1.570796, 2.126200],accel_mss,speed_ms,0,blend_radius_m)
    movel([0.553651, -1.230355, -2.658030, -0.824004, 1.570796, 2.124447],accel_mss,speed_ms,0,blend_radius_m)
    movel([0.551341, -1.232324, -2.657020, -0.823045, 1.570796, 2.122138],accel_mss,speed_ms,0,blend_radius_m)
    movel([0.548946, -1.234404, -2.655947, -0.822038, 1.570796, 2.119742],accel_mss,speed_ms,0,blend_radius_m)
    movel([0.546922, -1.235960, -2.655141, -0.821287, 1.570796, 2.117718],accel_mss,speed_ms,0,blend_radius_m)
    movel([0.542914, -1.238247, -2.653952, -0.820190, 1.570796, 2.113711],accel_mss,speed_ms,0,blend_radius_m)
    movel([0.539333, -1.239717, -2.653184, -0.819487, 1.570796, 2.110130],accel_mss,speed_ms,0,blend_radius_m)
    movel([0.536136, -1.240454, -2.652799, -0.819136, 1.570796, 2.106932],accel_mss,speed_ms,0,blend_radius_m)
    movel([0.533287, -1.240532, -2.652758, -0.819099, 1.570796, 2.104083],accel_mss,speed_ms,0,blend_radius_m)
    movel([0.530754, -1.240029, -2.653021, -0.819339, 1.570796, 2.101551],accel_mss,speed_ms,0,blend_radius_m)
    movel([0.528507, -1.239015, -2.653552, -0.819823, 1.570796, 2.099304],accel_mss,speed_ms,0,blend_radius_m)
    movel([0.526515, -1.237561, -2.654309, -0.820518, 1.570796, 2.097311],accel_mss,speed_ms,0,blend_radius_m)
    movel([0.524746, -1.235741, -2.655255, -0.821393, 1.570796, 2.095543],accel_mss,speed_ms,0,blend_radius_m)
    movel([0.521770, -1.231289, -2.657552, -0.823549, 1.570796, 2.092567],accel_mss,speed_ms,0,blend_radius_m)
    movel([0.519363, -1.226237, -2.660130, -0.826023, 1.570796, 2.090159],accel_mss,speed_ms,0,blend_radius_m)
    movel([0.515384, -1.216730, -2.664902, -0.830757, 1.570796, 2.086180],accel_mss,speed_ms,0,blend_radius_m)
    movel([0.513122, -1.212916, -2.666788, -0.832686, 1.570796, 2.083919],accel_mss,speed_ms,0,blend_radius_m)
    movel([0.509996, -1.208909, -2.668751, -0.834729, 1.570796, 2.080792],accel_mss,speed_ms,0,blend_radius_m)
    movel([0.506128, -1.204957, -2.670670, -0.836762, 1.570796, 2.076924],accel_mss,speed_ms,0,blend_radius_m)
    movel([0.501653, -1.201305, -2.672428, -0.838656, 1.570796, 2.072450],accel_mss,speed_ms,0,blend_radius_m)
    movel([0.496713, -1.198205, -2.673909, -0.840275, 1.570796, 2.067510],accel_mss,speed_ms,0,blend_radius_m)
    movel([0.491464, -1.195895, -2.675005, -0.841489, 1.570796, 2.062260],accel_mss,speed_ms,0,blend_radius_m)
    movel([0.486068, -1.194615, -2.675610, -0.842164, 1.570796, 2.056864],accel_mss,speed_ms,0,blend_radius_m)
    movel([0.483368, -1.194435, -2.675696, -0.842259, 1.570796, 2.054164],accel_mss,speed_ms,0,blend_radius_m)
    movel([0.480698, -1.194593, -2.675621, -0.842175, 1.570796, 2.051494],accel_mss,speed_ms,0,blend_radius_m)
    movel([0.477824, -1.195119, -2.675372, -0.841897, 1.570796, 2.048620],accel_mss,speed_ms,0,blend_radius_m)
    movel([0.474379, -1.196066, -2.674924, -0.841399, 1.570796, 2.045175],accel_mss,speed_ms,0,blend_radius_m)
    movel([0.470557, -1.197461, -2.674262, -0.840665, 1.570796, 2.041354],accel_mss,speed_ms,0,blend_radius_m)
    movel([0.466556, -1.199323, -2.673376, -0.839690, 1.570796, 2.037353],accel_mss,speed_ms,0,blend_radius_m)
    movel([0.462584, -1.201663, -2.672256, -0.838470, 1.570796, 2.033380],accel_mss,speed_ms,0,blend_radius_m)
    movel([0.458831, -1.204496, -2.670893, -0.837000, 1.570796, 2.029628],accel_mss,speed_ms,0,blend_radius_m)
    movel([0.455502, -1.207831, -2.669276, -0.835282, 1.570796, 2.026298],accel_mss,speed_ms,0,blend_radius_m)
    movel([0.454056, -1.209685, -2.668372, -0.834332, 1.570796, 2.024852],accel_mss,speed_ms,0,blend_radius_m)
    movel([0.452789, -1.211669, -2.667401, -0.833320, 1.570796, 2.023586],accel_mss,speed_ms,0,blend_radius_m)
    movel([0.451398, -1.214773, -2.665871, -0.831745, 1.570796, 2.022194],accel_mss,speed_ms,0,blend_radius_m)
    movel([0.450982, -1.217407, -2.664565, -0.830417, 1.570796, 2.021778],accel_mss,speed_ms,0,blend_radius_m)
    movel([0.451430, -1.219618, -2.663463, -0.829308, 1.570796, 2.022226],accel_mss,speed_ms,0,blend_radius_m)
    movel([0.452634, -1.221449, -2.662546, -0.828394, 1.570796, 2.023430],accel_mss,speed_ms,0,blend_radius_m)
    movel([0.454488, -1.222942, -2.661795, -0.827652, 1.570796, 2.025284],accel_mss,speed_ms,0,blend_radius_m)
    movel([0.456887, -1.224143, -2.661190, -0.827057, 1.570796, 2.027683],accel_mss,speed_ms,0,blend_radius_m)
    movel([0.459731, -1.225090, -2.660711, -0.826588, 1.570796, 2.030527],accel_mss,speed_ms,0,blend_radius_m)
    movel([0.462914, -1.225829, -2.660337, -0.826224, 1.570796, 2.033710],accel_mss,speed_ms,0,blend_radius_m)
    movel([0.469896, -1.226823, -2.659832, -0.825734, 1.570796, 2.040692],accel_mss,speed_ms,0,blend_radius_m)
    movel([0.477036, -1.227418, -2.659530, -0.825442, 1.570796, 2.047832],accel_mss,speed_ms,0,blend_radius_m)
    movel([0.483538, -1.227875, -2.659297, -0.825217, 1.570796, 2.054334],accel_mss,speed_ms,0,blend_radius_m)
    movel([0.488608, -1.228447, -2.659005, -0.824936, 1.570796, 2.059404],accel_mss,speed_ms,0,blend_radius_m)
    movel([0.500502, -1.230472, -2.657970, -0.823947, 1.570796, 2.071299],accel_mss,speed_ms,0,blend_radius_m)
    movel([0.506711, -1.231796, -2.657291, -0.823302, 1.570796, 2.077507],accel_mss,speed_ms,0,blend_radius_m)
    movel([0.511317, -1.233209, -2.656564, -0.822616, 1.570796, 2.082113],accel_mss,speed_ms,0,blend_radius_m)
    movel([0.512898, -1.234063, -2.656123, -0.822203, 1.570796, 2.083694],accel_mss,speed_ms,0,blend_radius_m)
    movel([0.514219, -1.235153, -2.655560, -0.821676, 1.570796, 2.085015],accel_mss,speed_ms,0,blend_radius_m)
    movel([0.516112, -1.237960, -2.654102, -0.820327, 1.570796, 2.086908],accel_mss,speed_ms,0,blend_radius_m)
    movel([0.517083, -1.241449, -2.652277, -0.818663, 1.570796, 2.087879],accel_mss,speed_ms,0,blend_radius_m)
    movel([0.517232, -1.245433, -2.650175, -0.816780, 1.570796, 2.088029],accel_mss,speed_ms,0,blend_radius_m)
    movel([0.516645, -1.249736, -2.647885, -0.814768, 1.570796, 2.087441],accel_mss,speed_ms,0,blend_radius_m)
    movel([0.515414, -1.254188, -2.645491, -0.812710, 1.570796, 2.086210],accel_mss,speed_ms,0,blend_radius_m)
    movel([0.513627, -1.258624, -2.643083, -0.810682, 1.570796, 2.084424],accel_mss,speed_ms,0,blend_radius_m)
    movel([0.511373, -1.262878, -2.640751, -0.808760, 1.570796, 2.082169],accel_mss,speed_ms,0,blend_radius_m)
    movel([0.507975, -1.267863, -2.637990, -0.806536, 1.570796, 2.078771],accel_mss,speed_ms,0,blend_radius_m)
    movel([0.506300, -1.269831, -2.636892, -0.805667, 1.570796, 2.077097],accel_mss,speed_ms,0,blend_radius_m)
    movel([0.504622, -1.271495, -2.635959, -0.804935, 1.570796, 2.075419],accel_mss,speed_ms,0,blend_radius_m)
    movel([0.502938, -1.272892, -2.635173, -0.804323, 1.570796, 2.073734],accel_mss,speed_ms,0,blend_radius_m)
    movel([0.501232, -1.274054, -2.634518, -0.803816, 1.570796, 2.072029],accel_mss,speed_ms,0,blend_radius_m)
    movel([0.497721, -1.275822, -2.633518, -0.803049, 1.570796, 2.068517],accel_mss,speed_ms,0,blend_radius_m)
    movel([0.494012, -1.277065, -2.632813, -0.802511, 1.570796, 2.064808],accel_mss,speed_ms,0,blend_radius_m)
    movel([0.490033, -1.278049, -2.632253, -0.802087, 1.570796, 2.060830],accel_mss,speed_ms,0,blend_radius_m)
    movel([0.480997, -1.280279, -2.630980, -0.801130, 1.570796, 2.051793],accel_mss,speed_ms,0,blend_radius_m)
    movel([0.480527, -1.280438, -2.630889, -0.801062, 1.570796, 2.051324],accel_mss,speed_ms,0,blend_radius_m)
    movel([0.480674, -1.280531, -2.630836, -0.801023, 1.570796, 2.051471],accel_mss,speed_ms,0,blend_radius_m)
    movel([0.482495, -1.280556, -2.630822, -0.801012, 1.570796, 2.053291],accel_mss,speed_ms,0,blend_radius_m)
    movel([0.489992, -1.280226, -2.631010, -0.801153, 1.570796, 2.060788],accel_mss,speed_ms,0,blend_radius_m)
    movel([0.502407, -1.279760, -2.631277, -0.801352, 1.570796, 2.073204],accel_mss,speed_ms,0,blend_radius_m)
    movel([0.495040, -1.283177, -2.629316, -0.799896, 1.570796, 2.065836],accel_mss,speed_ms,0,blend_radius_m)
    movel([0.486849, -1.286617, -2.627328, -0.798445, 1.570796, 2.057645],accel_mss,speed_ms,0,blend_radius_m)
    movel([0.478134, -1.290012, -2.625350, -0.797027, 1.570796, 2.048930],accel_mss,speed_ms,0,blend_radius_m)
    movel([0.469185, -1.293284, -2.623430, -0.795675, 1.570796, 2.039981],accel_mss,speed_ms,0,blend_radius_m)
    movel([0.451739, -1.299146, -2.619956, -0.793286, 1.570796, 2.022535],accel_mss,speed_ms,0,blend_radius_m)
    movel([0.443813, -1.301554, -2.618517, -0.792318, 1.570796, 2.014610],accel_mss,speed_ms,0,blend_radius_m)
    movel([0.436791, -1.303489, -2.617355, -0.791545, 1.570796, 2.007588],accel_mss,speed_ms,0,blend_radius_m)
    movel([0.426899, -1.309868, -2.613488, -0.789032, 1.570796, 1.997696],accel_mss,speed_ms,0,blend_radius_m)
    movel([0.416898, -1.316826, -2.609211, -0.786352, 1.570796, 1.987694],accel_mss,speed_ms,0,blend_radius_m)
    movel([0.396911, -1.331466, -2.600001, -0.780922, 1.570796, 1.967707],accel_mss,speed_ms,0,blend_radius_m)
    movel([0.387059, -1.338680, -2.595356, -0.778353, 1.570796, 1.957856],accel_mss,speed_ms,0,blend_radius_m)
    movel([0.377371, -1.345531, -2.590880, -0.775978, 1.570796, 1.948167],accel_mss,speed_ms,0,blend_radius_m)
    movel([0.367887, -1.351814, -2.586718, -0.773857, 1.570796, 1.938684],accel_mss,speed_ms,0,blend_radius_m)
    movel([0.358636, -1.357329, -2.583020, -0.772040, 1.570796, 1.929432],accel_mss,speed_ms,0,blend_radius_m)
    movel([0.355051, -1.359183, -2.581767, -0.771438, 1.570796, 1.925847],accel_mss,speed_ms,0,blend_radius_m)
    movel([0.351650, -1.360673, -2.580757, -0.770959, 1.570796, 1.922446],accel_mss,speed_ms,0,blend_radius_m)
    movel([0.348454, -1.361801, -2.579990, -0.770598, 1.570796, 1.919251],accel_mss,speed_ms,0,blend_radius_m)
    movel([0.345478, -1.362574, -2.579464, -0.770351, 1.570796, 1.916275],accel_mss,speed_ms,0,blend_radius_m)
    movel([0.342741, -1.362990, -2.579180, -0.770219, 1.570796, 1.913537],accel_mss,speed_ms,0,blend_radius_m)
    movel([0.340260, -1.363051, -2.579138, -0.770199, 1.570796, 1.911056],accel_mss,speed_ms,0,blend_radius_m)
    movel([0.338052, -1.362760, -2.579337, -0.770292, 1.570796, 1.908848],accel_mss,speed_ms,0,blend_radius_m)
    movel([0.336140, -1.362118, -2.579775, -0.770496, 1.570796, 1.906937],accel_mss,speed_ms,0,blend_radius_m)
    movel([0.334544, -1.361121, -2.580453, -0.770815, 1.570796, 1.905340],accel_mss,speed_ms,0,blend_radius_m)
    movel([0.333283, -1.359768, -2.581371, -0.771250, 1.570796, 1.904079],accel_mss,speed_ms,0,blend_radius_m)
    movel([0.332383, -1.358059, -2.582528, -0.771803, 1.570796, 1.903179],accel_mss,speed_ms,0,blend_radius_m)
    movel([0.331860, -1.355992, -2.583921, -0.772477, 1.570796, 1.902657],accel_mss,speed_ms,0,blend_radius_m)
    movel([0.331745, -1.353561, -2.585551, -0.773277, 1.570796, 1.902541],accel_mss,speed_ms,0,blend_radius_m)
    movel([0.332061, -1.350763, -2.587418, -0.774208, 1.570796, 1.902857],accel_mss,speed_ms,0,blend_radius_m)
    movel([0.332833, -1.347594, -2.589520, -0.775275, 1.570796, 1.903629],accel_mss,speed_ms,0,blend_radius_m)
    movel([0.334091, -1.344048, -2.591854, -0.776487, 1.570796, 1.904887],accel_mss,speed_ms,0,blend_radius_m)
    movel([0.336817, -1.345103, -2.591162, -0.776125, 1.570796, 1.907613],accel_mss,speed_ms,0,blend_radius_m)
    movel([0.338210, -1.345526, -2.590883, -0.775980, 1.570796, 1.909006],accel_mss,speed_ms,0,blend_radius_m)
    movel([0.339758, -1.345563, -2.590859, -0.775967, 1.570796, 1.910555],accel_mss,speed_ms,0,blend_radius_m)
    movel([0.341117, -1.345166, -2.591120, -0.776103, 1.570796, 1.911913],accel_mss,speed_ms,0,blend_radius_m)
    movel([0.342815, -1.344348, -2.591658, -0.776384, 1.570796, 1.913611],accel_mss,speed_ms,0,blend_radius_m)
    movel([0.347048, -1.341647, -2.593426, -0.777316, 1.570796, 1.917845],accel_mss,speed_ms,0,blend_radius_m)
    movel([0.352103, -1.337874, -2.595879, -0.778636, 1.570796, 1.922899],accel_mss,speed_ms,0,blend_radius_m)
    movel([0.357611, -1.333435, -2.598740, -0.780214, 1.570796, 1.928407],accel_mss,speed_ms,0,blend_radius_m)
    movel([0.368447, -1.324252, -2.604575, -0.783562, 1.570796, 1.939243],accel_mss,speed_ms,0,blend_radius_m)
